LIN {X 0,Y 262.031,Z 234.936,A -85,B 0,C 180,E1 -18600.13,E2 -18600.13} C_VEL
LIN {X 0,Y 263.652,Z 236.702,A -85,B 0,C 180,E1 -18600.64,E2 -18600.64} C_VEL
LIN {X 0,Y 266.299,Z 240.265,A -85,B 0,C 180,E1 -18601.481,E2 -18601.481} C_VEL
LIN {X 0,Y 273.867,Z 250.905,A -85,B 0,C 180,E1 -18603.757,E2 -18603.757} C_VEL
LIN {X 0,Y 283.8,Z 265.428,A -85,B 0,C 180,E1 -18606.486,E2 -18606.486} C_VEL
LIN {X 0,Y 294.582,Z 283.095,A -85,B 0,C 180,E1 -18609.207,E2 -18609.207} C_VEL
LIN {X 0,Y 301.927,Z 296.558,A -85,B 0,C 180,E1 -18610.957,E2 -18610.957} C_VEL
LIN {X 0,Y 295.132,Z 420.047,A -85,B 0,C 180,E1 -18613.929,E2 -18613.929} C_VEL
LIN {X 0,Y 293.462,Z 436.562,A -85,B 0,C 180,E1 -18614.548,E2 -18614.548} C_VEL
LIN {X 0,Y 291.234,Z 452.816,A -85,B 0,C 180,E1 -18615.411,E2 -18615.411} C_VEL
LIN {X 0,Y 288.511,Z 468.704,A -85,B 0,C 180,E1 -18616.529,E2 -18616.529} C_VEL
LIN {X 0,Y 285.326,Z 484.199,A -85,B 0,C 180,E1 -18617.914,E2 -18617.914} C_VEL
LIN {X 0,Y 281.734,Z 499.193,A -85,B 0,C 180,E1 -18619.58,E2 -18619.58} C_VEL
LIN {X 0,Y 277.76,Z 513.776,A -85,B 0,C 180,E1 -18621.583,E2 -18621.583} C_VEL
LIN {X 0,Y 273.902,Z 526.637,A -85,B 0,C 180,E1 -18623.739,E2 -18623.739} C_VEL
LIN {X 0,Y 269.966,Z 539.09,A -85,B 0,C 180,E1 -18626.268,E2 -18626.268} C_VEL
LIN {X 0,Y 266.441,Z 549.708,A -85,B 0,C 180,E1 -18628.866,E2 -18628.866} C_VEL
LIN {X 0,Y 263.361,Z 558.846,A -85,B 0,C 180,E1 -18631.529,E2 -18631.529} C_VEL
LIN {X 0,Y 260.495,Z 567.585,A -85,B 0,C 180,E1 -18634.642,E2 -18634.642} C_VEL
LIN {X 0,Y 258.128,Z 574.885,A -85,B 0,C 180,E1 -18637.824,E2 -18637.824} C_VEL
LIN {X 0,Y 256.372,Z 580.903,A -85,B 0,C 180,E1 -18641.063,E2 -18641.063} C_VEL
LIN {X 0,Y 255.118,Z 585.718,A -85,B 0,C 180,E1 -18644.355,E2 -18644.355} C_VEL
LIN {X 0,Y 254.241,Z 589.354,A -85,B 0,C 180,E1 -18647.702,E2 -18647.702} C_VEL
LIN {X 0,Y 253.781,Z 591.936,A -85,B 0,C 180,E1 -18651.1,E2 -18651.1} C_VEL
LIN {X 0,Y 253.539,Z 593.385,A -85,B 0,C 180,E1 -18654.568,E2 -18654.568} C_VEL
LIN {X 0,Y 253.58,Z 593.677,A -85,B 0,C 180,E1 -18658.108,E2 -18658.108} C_VEL
LIN {X 0,Y 253.912,Z 592.8,A -85,B 0,C 180,E1 -18661.728,E2 -18661.728} C_VEL
LIN {X 0,Y 254.646,Z 590.631,A -85,B 0,C 180,E1 -18665.42,E2 -18665.42} C_VEL
LIN {X 0,Y 255.905,Z 587.007,A -85,B 0,C 180,E1 -18669.171,E2 -18669.171} C_VEL
LIN {X 0,Y 257.498,Z 582.534,A -85,B 0,C 180,E1 -18672.53,E2 -18672.53} C_VEL
LIN {X 0,Y 259.761,Z 576.753,A -85,B 0,C 180,E1 -18675.906,E2 -18675.906} C_VEL
LIN {X 0,Y 262.976,Z 568.994,A -85,B 0,C 180,E1 -18679.453,E2 -18679.453} C_VEL
LIN {X 0,Y 266.826,Z 559.99,A -85,B 0,C 180,E1 -18682.714,E2 -18682.714} C_VEL
LIN {X 0,Y 270.696,Z 550.732,A -85,B 0,C 180,E1 -18685.442,E2 -18685.442} C_VEL
LIN {X 0,Y 275.191,Z 539.733,A -85,B 0,C 180,E1 -18688.118,E2 -18688.118} C_VEL
LIN {X 0,Y 279.707,Z 527.975,A -85,B 0,C 180,E1 -18690.481,E2 -18690.481} C_VEL
LIN {X 0,Y 284.292,Z 515.315,A -85,B 0,C 180,E1 -18692.58,E2 -18692.58} C_VEL
LIN {X 0,Y 288.929,Z 500.772,A -85,B 0,C 180,E1 -18694.558,E2 -18694.558} C_VEL
LIN {X 0,Y 292.994,Z 486.399,A -85,B 0,C 180,E1 -18696.132,E2 -18696.132} C_VEL
LIN {X 0,Y 296.725,Z 471.185,A -85,B 0,C 180,E1 -18697.474,E2 -18697.474} C_VEL
LIN {X 0,Y 299.894,Z 455.605,A -85,B 0,C 180,E1 -18698.562,E2 -18698.562} C_VEL
LIN {X 0,Y 302.505,Z 439.495,A -85,B 0,C 180,E1 -18699.42,E2 -18699.42} C_VEL
LIN {X 0,Y 304.524,Z 422.953,A -85,B 0,C 180,E1 -18700.038,E2 -18700.038} C_VEL
LIN {X 0,Y 307.609,Z 376.909,A -85,B 0,C 180,E1 -18701.178,E2 -18701.178} C_VEL
LIN {X 0,Y 307.523,Z 371.142,A -85,B 0,C 180,E1 -18701.419,E2 -18701.419} C_VEL
LIN {X 0,Y 305.147,Z 352.683,A -85,B 0,C 180,E1 -18702.697,E2 -18702.697} C_VEL
LIN {X 0,Y 305.135,Z 346.914,A -85,B 0,C 180,E1 -18702.932,E2 -18702.932} C_VEL
LIN {X 0,Y 307.991,Z 305.516,A -85,B 0,C 180,E1 -18703.919,E2 -18703.919} C_VEL
LIN {X 0,Y 303.595,Z 297.18,A -85,B 0,C 180,E1 -18705.428,E2 -18705.428} C_VEL
LIN {X 0,Y 298.427,Z 288.369,A -85,B 0,C 180,E1 -18707.322,E2 -18707.322} C_VEL
LIN {X 0,Y 292.108,Z 278.333,A -85,B 0,C 180,E1 -18709.899,E2 -18709.899} C_VEL
LIN {X 0,Y 288.353,Z 273.077,A -85,B 0,C 180,E1 -18711.591,E2 -18711.591} C_VEL
LIN {X 0,Y 285.651,Z 269.277,A -85,B 0,C 180,E1 -18712.934,E2 -18712.934} C_VEL
LIN {X 0,Y 282.696,Z 265.155,A -85,B 0,C 180,E1 -18714.519,E2 -18714.519} C_VEL
LIN {X 0,Y 279.765,Z 261.171,A -85,B 0,C 180,E1 -18716.295,E2 -18716.295} C_VEL
LIN {X 0,Y 276.977,Z 258.061,A -85,B 0,C 180,E1 -18718.139,E2 -18718.139} C_VEL
LIN {X 0,Y 275.666,Z 255.828,A -85,B 0,C 180,E1 -18719.178,E2 -18719.178} C_VEL
LIN {X 0,Y 273.124,Z 252.893,A -85,B 0,C 180,E1 -18721.366,E2 -18721.366} C_VEL
LIN {X 0,Y 272.174,Z 250.924,A -85,B 0,C 180,E1 -18722.397,E2 -18722.397} C_VEL
LIN {X 0,Y 269.161,Z 249.059,A -85,B 0,C 180,E1 -18725.995,E2 -18725.995} C_VEL
LIN {X 0,Y 267.506,Z 245.335,A -85,B 0,C 180,E1 -18730.597,E2 -18730.597} C_VEL
LIN {X 0,Y 267.455,Z 245.381,A -85,B 0,C 180,E1 -18734.829,E2 -18734.829} C_VEL
LIN {X 0,Y 269.144,Z 249.233,A -85,B 0,C 180,E1 -18739.645,E2 -18739.645} C_VEL
LIN {X 0,Y 271.78,Z 251.227,A -85,B 0,C 180,E1 -18742.917,E2 -18742.917} C_VEL
LIN {X 0,Y 273.593,Z 254.335,A -85,B 0,C 180,E1 -18744.799,E2 -18744.799} C_VEL
LIN {X 0,Y 276.027,Z 256.619,A -85,B 0,C 180,E1 -18746.766,E2 -18746.766} C_VEL
LIN {X 0,Y 278.612,Z 260.377,A -85,B 0,C 180,E1 -18748.638,E2 -18748.638} C_VEL
LIN {X 0,Y 280.09,Z 262,A -85,B 0,C 180,E1 -18749.576,E2 -18749.576} C_VEL
LIN {X 0,Y 284.743,Z 268.846,A -85,B 0,C 180,E1 -18752.279,E2 -18752.279} C_VEL
LIN {X 0,Y 288.411,Z 274.538,A -85,B 0,C 180,E1 -18754.152,E2 -18754.152} C_VEL
LIN {X 0,Y 292.215,Z 280.878,A -85,B 0,C 180,E1 -18755.911,E2 -18755.911} C_VEL
LIN {X 0,Y 297.089,Z 289.527,A -85,B 0,C 180,E1 -18757.956,E2 -18757.956} C_VEL
LIN {X 0,Y 302.308,Z 299.658,A -85,B 0,C 180,E1 -18759.962,E2 -18759.962} C_VEL
LIN {X 0,Y 307.047,Z 309.971,A -85,B 0,C 180,E1 -18761.661,E2 -18761.661} C_VEL
LIN {X 0,Y 307.643,Z 311.372,A -85,B 0,C 180,E1 -18761.87,E2 -18761.87} C_VEL
LIN {X 0,Y 301.033,Z 409.803,A -85,B 0,C 180,E1 -18764.234,E2 -18764.234} C_VEL
LIN {X 0,Y 299.152,Z 435.069,A -85,B 0,C 180,E1 -18764.894,E2 -18764.894} C_VEL
LIN {X 0,Y 296.911,Z 451.91,A -85,B 0,C 180,E1 -18765.521,E2 -18765.521} C_VEL
LIN {X 0,Y 293.976,Z 467.817,A -85,B 0,C 180,E1 -18766.347,E2 -18766.347} C_VEL
LIN {X 0,Y 290.572,Z 482.839,A -85,B 0,C 180,E1 -18767.374,E2 -18767.374} C_VEL
LIN {X 0,Y 286.439,Z 498.519,A -85,B 0,C 180,E1 -18768.747,E2 -18768.747} C_VEL
LIN {X 0,Y 281.831,Z 513.372,A -85,B 0,C 180,E1 -18770.353,E2 -18770.353} C_VEL
LIN {X 0,Y 277.266,Z 526.892,A -85,B 0,C 180,E1 -18772.176,E2 -18772.176} C_VEL
LIN {X 0,Y 272.027,Z 540.712,A -85,B 0,C 180,E1 -18774.459,E2 -18774.459} C_VEL
LIN {X 0,Y 267.105,Z 552.94,A -85,B 0,C 180,E1 -18776.955,E2 -18776.955} C_VEL
LIN {X 0,Y 262.933,Z 563.126,A -85,B 0,C 180,E1 -18779.48,E2 -18779.48} C_VEL
LIN {X 0,Y 259.086,Z 572.103,A -85,B 0,C 180,E1 -18782.101,E2 -18782.101} C_VEL
LIN {X 0,Y 254.99,Z 581.757,A -85,B 0,C 180,E1 -18785.581,E2 -18785.581} C_VEL
LIN {X 0,Y 251.535,Z 590.443,A -85,B 0,C 180,E1 -18789.559,E2 -18789.559} C_VEL
LIN {X 0,Y 249.09,Z 597.237,A -85,B 0,C 180,E1 -18793.612,E2 -18793.612} C_VEL
LIN {X 0,Y 247.847,Z 601.386,A -85,B 0,C 180,E1 -18796.889,E2 -18796.889} C_VEL
LIN {X 0,Y 247.104,Z 604.584,A -85,B 0,C 180,E1 -18800.175,E2 -18800.175} C_VEL
LIN {X 0,Y 246.856,Z 606.689,A -85,B 0,C 180,E1 -18803.462,E2 -18803.462} C_VEL
LIN {X 0,Y 246.839,Z 607.899,A -85,B 0,C 180,E1 -18806.736,E2 -18806.736} C_VEL
LIN {X 0,Y 246.983,Z 608.047,A -85,B 0,C 180,E1 -18810,E2 -18810} C_VEL
LIN {X 0,Y 246.868,Z 607.28,A -85,B 0,C 180,E1 -18813.264,E2 -18813.264} C_VEL
LIN {X 0,Y 246.859,Z 605.423,A -85,B 0,C 180,E1 -18816.539,E2 -18816.539} C_VEL
LIN {X 0,Y 247.096,Z 602.604,A -85,B 0,C 180,E1 -18819.826,E2 -18819.826} C_VEL
LIN {X 0,Y 248.074,Z 597.527,A -85,B 0,C 180,E1 -18823.934,E2 -18823.934} C_VEL
LIN {X 0,Y 249.357,Z 592.125,A -85,B 0,C 180,E1 -18827.214,E2 -18827.214} C_VEL
LIN {X 0,Y 251.252,Z 585.487,A -85,B 0,C 180,E1 -18830.466,E2 -18830.466} C_VEL
LIN {X 0,Y 253.657,Z 577.952,A -85,B 0,C 180,E1 -18833.512,E2 -18833.512} C_VEL
LIN {X 0,Y 257.031,Z 567.882,A -85,B 0,C 180,E1 -18836.818,E2 -18836.818} C_VEL
LIN {X 0,Y 260.52,Z 557.897,A -85,B 0,C 180,E1 -18839.494,E2 -18839.494} C_VEL
LIN {X 0,Y 263.756,Z 547.897,A -85,B 0,C 180,E1 -18841.783,E2 -18841.783} C_VEL
LIN {X 0,Y 267.797,Z 535.618,A -85,B 0,C 180,E1 -18844.122,E2 -18844.122} C_VEL
LIN {X 0,Y 271.945,Z 522.038,A -85,B 0,C 180,E1 -18846.24,E2 -18846.24} C_VEL
LIN {X 0,Y 275.628,Z 508.654,A -85,B 0,C 180,E1 -18847.962,E2 -18847.962} C_VEL
LIN {X 0,Y 279.266,Z 494.431,A -85,B 0,C 180,E1 -18849.453,E2 -18849.453} C_VEL
LIN {X 0,Y 282.538,Z 479.102,A -85,B 0,C 180,E1 -18850.765,E2 -18850.765} C_VEL
LIN {X 0,Y 285.543,Z 462.08,A -85,B 0,C 180,E1 -18851.884,E2 -18851.884} C_VEL
LIN {X 0,Y 287.982,Z 444.871,A -85,B 0,C 180,E1 -18852.686,E2 -18852.686} C_VEL
LIN {X 0,Y 289.505,Z 429.304,A -85,B 0,C 180,E1 -18853.181,E2 -18853.181} C_VEL
LIN {X 0,Y 296.362,Z 306.373,A -85,B 0,C 180,E1 -18856.178,E2 -18856.178} C_VEL
LIN {X 0,Y 288.532,Z 290.028,A -85,B 0,C 180,E1 -18858.18,E2 -18858.18} C_VEL
LIN {X 0,Y 280.5,Z 274.97,A -85,B 0,C 180,E1 -18860.348,E2 -18860.348} C_VEL
LIN {X 0,Y 272.954,Z 261.95,A -85,B 0,C 180,E1 -18862.512,E2 -18862.512} C_VEL
LIN {X 0,Y 266.916,Z 252.198,A -85,B 0,C 180,E1 -18864.362,E2 -18864.362} C_VEL
LIN {X 0,Y 262.167,Z 245.051,A -85,B 0,C 180,E1 -18865.891,E2 -18865.891} C_VEL
LIN {X 0,Y 259.448,Z 241.346,A -85,B 0,C 180,E1 -18866.791,E2 -18866.791} C_VEL
LIN {X 0,Y 256.707,Z 237.544,A -85,B 0,C 180,E1 -18867.735,E2 -18867.735} C_VEL
LIN {X 0,Y 253.618,Z 233.906,A -85,B 0,C 180,E1 -18868.812,E2 -18868.812} C_VEL
LIN {X 0,Y 252.501,Z 232.01,A -85,B 0,C 180,E1 -18869.24,E2 -18869.24} C_VEL
LIN {X 0,Y 250.243,Z 229.914,A -85,B 0,C 180,E1 -18870.039,E2 -18870.039} C_VEL
LIN {X 0,Y 249.171,Z 227.301,A -85,B 0,C 180,E1 -18870.514,E2 -18870.514} C_VEL
LIN {X 0,Y 249.076,Z 226.767,A -85,B 0,C 180,E1 -18870.596,E2 -18870.596} C_VEL
LIN {X 0,Y 249.15,Z 226.733,A -85,B 0,C 180,E1 -18874.969,E2 -18874.969} C_VEL
LIN {X 0,Y 249.093,Z 226.751,A -85,B 0,C 180,E1 -18878.602,E2 -18878.602} C_VEL
LIN {X 0,Y 249.195,Z 226.752,A -85,B 0,C 180,E1 -18883.619,E2 -18883.619} C_VEL
LIN {X 0,Y 249.224,Z 226.704,A -85,B 0,C 180,E1 -18888.615,E2 -18888.615} C_VEL
LIN {X 0,Y 249.441,Z 226.724,A -85,B 0,C 180,E1 -18891.902,E2 -18891.902} C_VEL
LIN {X 0,Y 249.287,Z 226.704,A -85,B 0,C 180,E1 -18895.148,E2 -18895.148} C_VEL
LIN {X 0,Y 249.673,Z 226.648,A -85,B 0,C 180,E1 -18898.387,E2 -18898.387} C_VEL
LIN {X 0,Y 249.674,Z 226.697,A -85,B 0,C 180,E1 -18901.613,E2 -18901.613} C_VEL
LIN {X 0,Y 249.439,Z 226.705,A -85,B 0,C 180,E1 -18906.718,E2 -18906.718} C_VEL
LIN {X 0,Y 249.343,Z 226.728,A -85,B 0,C 180,E1 -18909.736,E2 -18909.736} C_VEL
LIN {X 0,Y 249.205,Z 226.752,A -85,B 0,C 180,E1 -18914.703,E2 -18914.703} C_VEL
LIN {X 0,Y 249.139,Z 226.734,A -85,B 0,C 180,E1 -18918.077,E2 -18918.077} C_VEL
LIN {X 0,Y 249.087,Z 226.767,A -85,B 0,C 180,E1 -18921.518,E2 -18921.518} C_VEL
LIN {X 0,Y 249.131,Z 226.735,A -85,B 0,C 180,E1 -18925.482,E2 -18925.482} C_VEL
LIN {X 0,Y 249.087,Z 226.771,A -85,B 0,C 180,E1 -18928.995,E2 -18928.995} C_VEL
LIN {X 0,Y 249.03,Z 226.751,A -85,B 0,C 180,E1 -18932.426,E2 -18932.426} C_VEL
LIN {X 0,Y 249.047,Z 226.766,A -85,B 0,C 180,E1 -18936.342,E2 -18936.342} C_VEL
LIN {X 0,Y 249.006,Z 226.779,A -85,B 0,C 180,E1 -18940.478,E2 -18940.478} C_VEL
LIN {X 0,Y 248.992,Z 226.766,A -85,B 0,C 180,E1 -18944.881,E2 -18944.881} C_VEL
LIN {X 0,Y 249.015,Z 226.773,A -85,B 0,C 180,E1 -18947.363,E2 -18947.363} C_VEL
LIN {X 0,Y 249.043,Z 226.769,A -85,B 0,C 180,E1 -18952.2,E2 -18952.2} C_VEL
LIN {X 0,Y 249.04,Z 226.774,A -85,B 0,C 180,E1 -18955.931,E2 -18955.931} C_VEL
LIN {X 0,Y 249.82,Z 229.243,A -85,B 0,C 180,E1 -18956.312,E2 -18956.312} C_VEL
LIN {X 0,Y 251.534,Z 231.358,A -85,B 0,C 180,E1 -18956.952,E2 -18956.952} C_VEL
LIN {X 0,Y 252.919,Z 232.5,A -85,B 0,C 180,E1 -18957.431,E2 -18957.431} C_VEL
LIN {X 0,Y 254.879,Z 235.654,A -85,B 0,C 180,E1 -18958.17,E2 -18958.17} C_VEL
LIN {X 0,Y 256.812,Z 237.703,A -85,B 0,C 180,E1 -18958.826,E2 -18958.826} C_VEL
LIN {X 0,Y 259.44,Z 241.277,A -85,B 0,C 180,E1 -18959.724,E2 -18959.724} C_VEL
LIN {X 0,Y 264.351,Z 247.934,A -85,B 0,C 180,E1 -18961.322,E2 -18961.322} C_VEL
LIN {X 0,Y 271.132,Z 257.534,A -85,B 0,C 180,E1 -18963.396,E2 -18963.396} C_VEL
LIN {X 0,Y 280.204,Z 271.03,A -85,B 0,C 180,E1 -18965.95,E2 -18965.95} C_VEL
LIN {X 0,Y 290.389,Z 287.903,A -85,B 0,C 180,E1 -18968.604,E2 -18968.604} C_VEL
LIN {X 0,Y 296.481,Z 299.015,A -85,B 0,C 180,E1 -18970.096,E2 -18970.096} C_VEL
LIN {X 0,Y 289.59,Z 420.591,A -85,B 0,C 180,E1 -18973.068,E2 -18973.068} C_VEL
LIN {X 0,Y 287.767,Z 437.863,A -85,B 0,C 180,E1 -18973.734,E2 -18973.734} C_VEL
LIN {X 0,Y 285.368,Z 454.472,A -85,B 0,C 180,E1 -18974.649,E2 -18974.649} C_VEL
LIN {X 0,Y 282.549,Z 470.029,A -85,B 0,C 180,E1 -18975.781,E2 -18975.781} C_VEL
LIN {X 0,Y 279.48,Z 484.488,A -85,B 0,C 180,E1 -18977.104,E2 -18977.104} C_VEL
LIN {X 0,Y 275.759,Z 499.477,A -85,B 0,C 180,E1 -18978.794,E2 -18978.794} C_VEL
LIN {X 0,Y 271.899,Z 513.198,A -85,B 0,C 180,E1 -18980.703,E2 -18980.703} C_VEL
LIN {X 0,Y 267.953,Z 525.923,A -85,B 0,C 180,E1 -18982.843,E2 -18982.843} C_VEL
LIN {X 0,Y 263.832,Z 538.529,A -85,B 0,C 180,E1 -18985.416,E2 -18985.416} C_VEL
LIN {X 0,Y 260.187,Z 549.178,A -85,B 0,C 180,E1 -18988.039,E2 -18988.039} C_VEL
LIN {X 0,Y 256.875,Z 558.489,A -85,B 0,C 180,E1 -18990.783,E2 -18990.783} C_VEL
LIN {X 0,Y 254.101,Z 566.572,A -85,B 0,C 180,E1 -18993.676,E2 -18993.676} C_VEL
LIN {X 0,Y 251.966,Z 573.039,A -85,B 0,C 180,E1 -18996.405,E2 -18996.405} C_VEL
LIN {X 0,Y 249.78,Z 579.919,A -85,B 0,C 180,E1 -19000.008,E2 -19000.008} C_VEL
LIN {X 0,Y 248.437,Z 584.554,A -85,B 0,C 180,E1 -19003.079,E2 -19003.079} C_VEL
LIN {X 0,Y 247.423,Z 588.606,A -85,B 0,C 180,E1 -19006.501,E2 -19006.501} C_VEL
LIN {X 0,Y 246.813,Z 591.473,A -85,B 0,C 180,E1 -19010.003,E2 -19010.003} C_VEL
LIN {X 0,Y 246.5,Z 593.256,A -85,B 0,C 180,E1 -19013.525,E2 -19013.525} C_VEL
LIN {X 0,Y 246.47,Z 593.959,A -85,B 0,C 180,E1 -19017.143,E2 -19017.143} C_VEL
LIN {X 0,Y 246.772,Z 593.275,A -85,B 0,C 180,E1 -19021.308,E2 -19021.308} C_VEL
LIN {X 0,Y 247.347,Z 591.61,A -85,B 0,C 180,E1 -19024.629,E2 -19024.629} C_VEL
LIN {X 0,Y 248.521,Z 588.471,A -85,B 0,C 180,E1 -19028.472,E2 -19028.472} C_VEL
LIN {X 0,Y 250.303,Z 583.834,A -85,B 0,C 180,E1 -19032.365,E2 -19032.365} C_VEL
LIN {X 0,Y 252.908,Z 577.541,A -85,B 0,C 180,E1 -19036.26,E2 -19036.26} C_VEL
LIN {X 0,Y 255.621,Z 571.302,A -85,B 0,C 180,E1 -19039.275,E2 -19039.275} C_VEL
LIN {X 0,Y 259.171,Z 563.406,A -85,B 0,C 180,E1 -19042.407,E2 -19042.407} C_VEL
LIN {X 0,Y 263.047,Z 554.718,A -85,B 0,C 180,E1 -19045.24,E2 -19045.24} C_VEL
LIN {X 0,Y 267.499,Z 544.525,A -85,B 0,C 180,E1 -19047.951,E2 -19047.951} C_VEL
LIN {X 0,Y 272.168,Z 533.037,A -85,B 0,C 180,E1 -19050.494,E2 -19050.494} C_VEL
LIN {X 0,Y 277.286,Z 519.862,A -85,B 0,C 180,E1 -19052.857,E2 -19052.857} C_VEL
LIN {X 0,Y 281.815,Z 506.845,A -85,B 0,C 180,E1 -19054.785,E2 -19054.785} C_VEL
LIN {X 0,Y 286.126,Z 493.17,A -85,B 0,C 180,E1 -19056.437,E2 -19056.437} C_VEL
LIN {X 0,Y 290.151,Z 478.375,A -85,B 0,C 180,E1 -19057.891,E2 -19057.891} C_VEL
LIN {X 0,Y 293.792,Z 462.5,A -85,B 0,C 180,E1 -19059.135,E2 -19059.135} C_VEL
LIN {X 0,Y 296.806,Z 446.047,A -85,B 0,C 180,E1 -19060.131,E2 -19060.131} C_VEL
LIN {X 0,Y 299.107,Z 430.324,A -85,B 0,C 180,E1 -19060.814,E2 -19060.814} C_VEL
LIN {X 0,Y 300.702,Z 413.397,A -85,B 0,C 180,E1 -19061.331,E2 -19061.331} C_VEL
LIN {X 0,Y 305.135,Z 346.914,A -85,B 0,C 180,E1 -19062.932,E2 -19062.932} C_VEL
LIN {X 0,Y 305.117,Z 341.14,A -85,B 0,C 180,E1 -19063.172,E2 -19063.172} C_VEL
LIN {X 0,Y 302.957,Z 322.696,A -85,B 0,C 180,E1 -19064.495,E2 -19064.495} C_VEL
LIN {X 0,Y 303.017,Z 316.921,A -85,B 0,C 180,E1 -19064.727,E2 -19064.727} C_VEL
LIN {X 0,Y 303.577,Z 308.469,A -85,B 0,C 180,E1 -19064.943,E2 -19064.943} C_VEL
LIN {X 0,Y 297.727,Z 297.627,A -85,B 0,C 180,E1 -19067.094,E2 -19067.094} C_VEL
LIN {X 0,Y 291.284,Z 287.028,A -85,B 0,C 180,E1 -19069.722,E2 -19069.722} C_VEL
LIN {X 0,Y 287.001,Z 280.473,A -85,B 0,C 180,E1 -19071.689,E2 -19071.689} C_VEL
LIN {X 0,Y 283.314,Z 275.274,A -85,B 0,C 180,E1 -19073.567,E2 -19073.567} C_VEL
LIN {X 0,Y 280.767,Z 271.594,A -85,B 0,C 180,E1 -19075.004,E2 -19075.004} C_VEL
LIN {X 0,Y 277.936,Z 267.662,A -85,B 0,C 180,E1 -19076.788,E2 -19076.788} C_VEL
LIN {X 0,Y 275.207,Z 264.392,A -85,B 0,C 180,E1 -19078.691,E2 -19078.691} C_VEL
LIN {X 0,Y 274.093,Z 262.494,A -85,B 0,C 180,E1 -19079.611,E2 -19079.611} C_VEL
LIN {X 0,Y 271.623,Z 259.443,A -85,B 0,C 180,E1 -19081.853,E2 -19081.853} C_VEL
LIN {X 0,Y 270.795,Z 257.779,A -85,B 0,C 180,E1 -19082.788,E2 -19082.788} C_VEL
LIN {X 0,Y 268.104,Z 256.047,A -85,B 0,C 180,E1 -19086.14,E2 -19086.14} C_VEL
LIN {X 0,Y 266.541,Z 252.403,A -85,B 0,C 180,E1 -19090.636,E2 -19090.636} C_VEL
LIN {X 0,Y 266.469,Z 252.375,A -85,B 0,C 180,E1 -19094.639,E2 -19094.639} C_VEL
LIN {X 0,Y 268.102,Z 256.239,A -85,B 0,C 180,E1 -19099.525,E2 -19099.525} C_VEL
LIN {X 0,Y 270.449,Z 258.043,A -85,B 0,C 180,E1 -19102.554,E2 -19102.554} C_VEL
LIN {X 0,Y 272.334,Z 261.239,A -85,B 0,C 180,E1 -19104.565,E2 -19104.565} C_VEL
LIN {X 0,Y 274.434,Z 263.232,A -85,B 0,C 180,E1 -19106.324,E2 -19106.324} C_VEL
LIN {X 0,Y 277.07,Z 267.119,A -85,B 0,C 180,E1 -19108.308,E2 -19108.308} C_VEL
LIN {X 0,Y 278.306,Z 268.529,A -85,B 0,C 180,E1 -19109.118,E2 -19109.118} C_VEL
LIN {X 0,Y 282.522,Z 274.891,A -85,B 0,C 180,E1 -19111.685,E2 -19111.685} C_VEL
LIN {X 0,Y 286.095,Z 280.674,A -85,B 0,C 180,E1 -19113.589,E2 -19113.589} C_VEL
LIN {X 0,Y 289.17,Z 285.918,A -85,B 0,C 180,E1 -19115.088,E2 -19115.088} C_VEL
LIN {X 0,Y 293.972,Z 294.702,A -85,B 0,C 180,E1 -19117.221,E2 -19117.221} C_VEL
LIN {X 0,Y 299.004,Z 304.731,A -85,B 0,C 180,E1 -19119.256,E2 -19119.256} C_VEL
LIN {X 0,Y 303.342,Z 314.363,A -85,B 0,C 180,E1 -19120.882,E2 -19120.882} C_VEL
LIN {X 0,Y 294.908,Z 432.361,A -85,B 0,C 180,E1 -19123.756,E2 -19123.756} C_VEL
LIN {X 0,Y 292.717,Z 449.242,A -85,B 0,C 180,E1 -19124.365,E2 -19124.365} C_VEL
LIN {X 0,Y 289.958,Z 464.391,A -85,B 0,C 180,E1 -19125.107,E2 -19125.107} C_VEL
LIN {X 0,Y 286.429,Z 480.071,A -85,B 0,C 180,E1 -19126.121,E2 -19126.121} C_VEL
LIN {X 0,Y 282.62,Z 494.63,A -85,B 0,C 180,E1 -19127.342,E2 -19127.342} C_VEL
LIN {X 0,Y 277.936,Z 509.588,A -85,B 0,C 180,E1 -19128.896,E2 -19128.896} C_VEL
LIN {X 0,Y 273.365,Z 522.759,A -85,B 0,C 180,E1 -19130.595,E2 -19130.595} C_VEL
LIN {X 0,Y 268.623,Z 535.26,A -85,B 0,C 180,E1 -19132.535,E2 -19132.535} C_VEL
LIN {X 0,Y 264.064,Z 546.425,A -85,B 0,C 180,E1 -19134.63,E2 -19134.63} C_VEL
LIN {X 0,Y 259.165,Z 557.798,A -85,B 0,C 180,E1 -19137.209,E2 -19137.209} C_VEL
LIN {X 0,Y 254.369,Z 568.531,A -85,B 0,C 180,E1 -19140.178,E2 -19140.178} C_VEL
LIN {X 0,Y 250.246,Z 577.75,A -85,B 0,C 180,E1 -19143.299,E2 -19143.299} C_VEL
LIN {X 0,Y 246.88,Z 585.475,A -85,B 0,C 180,E1 -19146.514,E2 -19146.514} C_VEL
LIN {X 0,Y 244.195,Z 591.877,A -85,B 0,C 180,E1 -19149.797,E2 -19149.797} C_VEL
LIN {X 0,Y 242.119,Z 597.41,A -85,B 0,C 180,E1 -19153.313,E2 -19153.313} C_VEL
LIN {X 0,Y 240.864,Z 601.283,A -85,B 0,C 180,E1 -19156.502,E2 -19156.502} C_VEL
LIN {X 0,Y 240.04,Z 604.442,A -85,B 0,C 180,E1 -19159.883,E2 -19159.883} C_VEL
LIN {X 0,Y 239.767,Z 606.529,A -85,B 0,C 180,E1 -19163.267,E2 -19163.267} C_VEL
LIN {X 0,Y 239.744,Z 607.702,A -85,B 0,C 180,E1 -19166.639,E2 -19166.639} C_VEL
LIN {X 0,Y 239.913,Z 607.831,A -85,B 0,C 180,E1 -19170,E2 -19170} C_VEL
LIN {X 0,Y 239.774,Z 607.025,A -85,B 0,C 180,E1 -19173.361,E2 -19173.361} C_VEL
LIN {X 0,Y 239.821,Z 606.225,A -85,B 0,C 180,E1 -19175.044,E2 -19175.044} C_VEL
LIN {X 0,Y 239.872,Z 603.837,A -85,B 0,C 180,E1 -19178.424,E2 -19178.424} C_VEL
LIN {X 0,Y 240.328,Z 600.46,A -85,B 0,C 180,E1 -19181.812,E2 -19181.812} C_VEL
LIN {X 0,Y 241.675,Z 594.851,A -85,B 0,C 180,E1 -19185.88,E2 -19185.88} C_VEL
LIN {X 0,Y 243.38,Z 588.545,A -85,B 0,C 180,E1 -19189.395,E2 -19189.395} C_VEL
LIN {X 0,Y 245.775,Z 581.2,A -85,B 0,C 180,E1 -19192.708,E2 -19192.708} C_VEL
LIN {X 0,Y 248.772,Z 572.38,A -85,B 0,C 180,E1 -19195.969,E2 -19195.969} C_VEL
LIN {X 0,Y 252.593,Z 561.814,A -85,B 0,C 180,E1 -19199.138,E2 -19199.138} C_VEL
LIN {X 0,Y 256.238,Z 551.194,A -85,B 0,C 180,E1 -19201.761,E2 -19201.761} C_VEL
LIN {X 0,Y 260.141,Z 539.855,A -85,B 0,C 180,E1 -19204.096,E2 -19204.096} C_VEL
LIN {X 0,Y 264.271,Z 527.153,A -85,B 0,C 180,E1 -19206.279,E2 -19206.279} C_VEL
LIN {X 0,Y 268.62,Z 512.782,A -85,B 0,C 180,E1 -19208.289,E2 -19208.289} C_VEL
LIN {X 0,Y 272.422,Z 498.392,A -85,B 0,C 180,E1 -19209.921,E2 -19209.921} C_VEL
LIN {X 0,Y 276.057,Z 482.886,A -85,B 0,C 180,E1 -19211.325,E2 -19211.325} C_VEL
LIN {X 0,Y 279.119,Z 466.976,A -85,B 0,C 180,E1 -19212.463,E2 -19212.463} C_VEL
LIN {X 0,Y 281.564,Z 451.74,A -85,B 0,C 180,E1 -19213.286,E2 -19213.286} C_VEL
LIN {X 0,Y 283.655,Z 434.645,A -85,B 0,C 180,E1 -19213.927,E2 -19213.927} C_VEL
LIN {X 0,Y 287.302,Z 371.522,A -85,B 0,C 180,E1 -19215.53,E2 -19215.53} C_VEL
LIN {X 0,Y 290.939,Z 308.736,A -85,B 0,C 180,E1 -19217.067,E2 -19217.067} C_VEL
LIN {X 0,Y 283.914,Z 293.977,A -85,B 0,C 180,E1 -19218.934,E2 -19218.934} C_VEL
LIN {X 0,Y 276.164,Z 279.314,A -85,B 0,C 180,E1 -19221.1,E2 -19221.1} C_VEL
LIN {X 0,Y 269.039,Z 266.863,A -85,B 0,C 180,E1 -19223.226,E2 -19223.226} C_VEL
LIN {X 0,Y 263.188,Z 257.265,A -85,B 0,C 180,E1 -19225.079,E2 -19225.079} C_VEL
LIN {X 0,Y 258.352,Z 249.977,A -85,B 0,C 180,E1 -19226.69,E2 -19226.69} C_VEL
LIN {X 0,Y 255.752,Z 246.482,A -85,B 0,C 180,E1 -19227.579,E2 -19227.579} C_VEL
LIN {X 0,Y 252.776,Z 242.472,A -85,B 0,C 180,E1 -19228.638,E2 -19228.638} C_VEL
LIN {X 0,Y 250.118,Z 238.942,A -85,B 0,C 180,E1 -19229.617,E2 -19229.617} C_VEL
LIN {X 0,Y 248.959,Z 237.619,A -85,B 0,C 180,E1 -19230.046,E2 -19230.046} C_VEL
LIN {X 0,Y 246.642,Z 234.687,A -85,B 0,C 180,E1 -19230.944,E2 -19230.944} C_VEL
LIN {X 0,Y 245.802,Z 233.041,A -85,B 0,C 180,E1 -19231.309,E2 -19231.309} C_VEL
LIN {X 0,Y 243.556,Z 231.25,A -85,B 0,C 180,E1 -19232.154,E2 -19232.154} C_VEL
LIN {X 0,Y 242.234,Z 228.656,A -85,B 0,C 180,E1 -19232.751,E2 -19232.751} C_VEL
LIN {X 0,Y 242.037,Z 227.621,A -85,B 0,C 180,E1 -19232.903,E2 -19232.903} C_VEL
LIN {X 0,Y 242.056,Z 227.63,A -85,B 0,C 180,E1 -19236.016,E2 -19236.016} C_VEL
LIN {X 0,Y 242.025,Z 227.614,A -85,B 0,C 180,E1 -19239.607,E2 -19239.607} C_VEL
LIN {X 0,Y 242.115,Z 227.628,A -85,B 0,C 180,E1 -19243.316,E2 -19243.316} C_VEL
LIN {X 0,Y 242.134,Z 227.6,A -85,B 0,C 180,E1 -19246.573,E2 -19246.573} C_VEL
LIN {X 0,Y 242.388,Z 227.599,A -85,B 0,C 180,E1 -19251.664,E2 -19251.664} C_VEL
LIN {X 0,Y 242.415,Z 227.597,A -85,B 0,C 180,E1 -19253.341,E2 -19253.341} C_VEL
LIN {X 0,Y 242.633,Z 227.523,A -85,B 0,C 180,E1 -19258.34,E2 -19258.34} C_VEL
LIN {X 0,Y 242.635,Z 227.574,A -85,B 0,C 180,E1 -19261.66,E2 -19261.66} C_VEL
LIN {X 0,Y 242.42,Z 227.58,A -85,B 0,C 180,E1 -19266.69,E2 -19266.69} C_VEL
LIN {X 0,Y 242.267,Z 227.604,A -85,B 0,C 180,E1 -19270.024,E2 -19270.024} C_VEL
LIN {X 0,Y 242.166,Z 227.63,A -85,B 0,C 180,E1 -19275.141,E2 -19275.141} C_VEL
LIN {X 0,Y 242.072,Z 227.611,A -85,B 0,C 180,E1 -19278.624,E2 -19278.624} C_VEL
LIN {X 0,Y 242.013,Z 227.651,A -85,B 0,C 180,E1 -19282.18,E2 -19282.18} C_VEL
LIN {X 0,Y 242.066,Z 227.615,A -85,B 0,C 180,E1 -19285.838,E2 -19285.838} C_VEL
LIN {X 0,Y 242.031,Z 227.645,A -85,B 0,C 180,E1 -19289.58,E2 -19289.58} C_VEL
LIN {X 0,Y 241.98,Z 227.638,A -85,B 0,C 180,E1 -19293.493,E2 -19293.493} C_VEL
LIN {X 0,Y 241.988,Z 227.631,A -85,B 0,C 180,E1 -19297.582,E2 -19297.582} C_VEL
LIN {X 0,Y 241.933,Z 227.656,A -85,B 0,C 180,E1 -19301.923,E2 -19301.923} C_VEL
LIN {X 0,Y 241.932,Z 227.663,A -85,B 0,C 180,E1 -19306.572,E2 -19306.572} C_VEL
LIN {X 0,Y 241.995,Z 227.654,A -85,B 0,C 180,E1 -19311.64,E2 -19311.64} C_VEL
LIN {X 0,Y 242.007,Z 227.631,A -85,B 0,C 180,E1 -19313.613,E2 -19313.613} C_VEL
LIN {X 0,Y 242.841,Z 230.251,A -85,B 0,C 180,E1 -19314.065,E2 -19314.065} C_VEL
LIN {X 0,Y 244.62,Z 232.316,A -85,B 0,C 180,E1 -19314.788,E2 -19314.788} C_VEL
LIN {X 0,Y 246.005,Z 233.437,A -85,B 0,C 180,E1 -19315.309,E2 -19315.309} C_VEL
LIN {X 0,Y 247.819,Z 236.494,A -85,B 0,C 180,E1 -19316.056,E2 -19316.056} C_VEL
LIN {X 0,Y 250.001,Z 238.742,A -85,B 0,C 180,E1 -19316.854,E2 -19316.854} C_VEL
LIN {X 0,Y 252.623,Z 242.292,A -85,B 0,C 180,E1 -19317.827,E2 -19317.827} C_VEL
LIN {X 0,Y 253.937,Z 243.955,A -85,B 0,C 180,E1 -19318.298,E2 -19318.298} C_VEL
LIN {X 0,Y 258.355,Z 249.931,A -85,B 0,C 180,E1 -19319.828,E2 -19319.828} C_VEL
LIN {X 0,Y 263.589,Z 257.098,A -85,B 0,C 180,E1 -19321.533,E2 -19321.533} C_VEL
LIN {X 0,Y 273.699,Z 272.015,A -85,B 0,C 180,E1 -19324.577,E2 -19324.577} C_VEL
LIN {X 0,Y 283.097,Z 287.351,A -85,B 0,C 180,E1 -19327.163,E2 -19327.163} C_VEL
LIN {X 0,Y 291.075,Z 301.655,A -85,B 0,C 180,E1 -19329.218,E2 -19329.218} C_VEL
LIN {X 0,Y 284.114,Z 420.909,A -85,B 0,C 180,E1 -19332.175,E2 -19332.175} C_VEL
LIN {X 0,Y 282.224,Z 438.164,A -85,B 0,C 180,E1 -19332.846,E2 -19332.846} C_VEL
LIN {X 0,Y 279.77,Z 454.714,A -85,B 0,C 180,E1 -19333.771,E2 -19333.771} C_VEL
LIN {X 0,Y 276.905,Z 470.097,A -85,B 0,C 180,E1 -19334.903,E2 -19334.903} C_VEL
LIN {X 0,Y 273.682,Z 484.76,A -85,B 0,C 180,E1 -19336.259,E2 -19336.259} C_VEL
LIN {X 0,Y 269.831,Z 499.758,A -85,B 0,C 180,E1 -19337.973,E2 -19337.973} C_VEL
LIN {X 0,Y 265.843,Z 513.477,A -85,B 0,C 180,E1 -19339.913,E2 -19339.913} C_VEL
LIN {X 0,Y 261.444,Z 527.177,A -85,B 0,C 180,E1 -19342.275,E2 -19342.275} C_VEL
LIN {X 0,Y 257.211,Z 539.611,A -85,B 0,C 180,E1 -19344.905,E2 -19344.905} C_VEL
LIN {X 0,Y 253.197,Z 550.784,A -85,B 0,C 180,E1 -19347.778,E2 -19347.778} C_VEL
LIN {X 0,Y 249.644,Z 560.484,A -85,B 0,C 180,E1 -19350.806,E2 -19350.806} C_VEL
LIN {X 0,Y 246.6,Z 569.05,A -85,B 0,C 180,E1 -19354.066,E2 -19354.066} C_VEL
LIN {X 0,Y 244.088,Z 576.205,A -85,B 0,C 180,E1 -19357.444,E2 -19357.444} C_VEL
LIN {X 0,Y 242.206,Z 582.028,A -85,B 0,C 180,E1 -19360.871,E2 -19360.871} C_VEL
LIN {X 0,Y 240.923,Z 586.701,A -85,B 0,C 180,E1 -19364.356,E2 -19364.356} C_VEL
LIN {X 0,Y 240.211,Z 589.413,A -85,B 0,C 180,E1 -19367.012,E2 -19367.012} C_VEL
LIN {X 0,Y 239.631,Z 592.137,A -85,B 0,C 180,E1 -19370.605,E2 -19370.605} C_VEL
LIN {X 0,Y 239.366,Z 593.735,A -85,B 0,C 180,E1 -19374.469,E2 -19374.469} C_VEL
LIN {X 0,Y 239.428,Z 594.104,A -85,B 0,C 180,E1 -19378.286,E2 -19378.286} C_VEL
LIN {X 0,Y 239.731,Z 593.405,A -85,B 0,C 180,E1 -19381.849,E2 -19381.849} C_VEL
LIN {X 0,Y 240.518,Z 591.324,A -85,B 0,C 180,E1 -19385.76,E2 -19385.76} C_VEL
LIN {X 0,Y 241.926,Z 587.874,A -85,B 0,C 180,E1 -19389.724,E2 -19389.724} C_VEL
LIN {X 0,Y 243.989,Z 582.912,A -85,B 0,C 180,E1 -19393.733,E2 -19393.733} C_VEL
LIN {X 0,Y 246.126,Z 578.114,A -85,B 0,C 180,E1 -19396.74,E2 -19396.74} C_VEL
LIN {X 0,Y 249.321,Z 571.189,A -85,B 0,C 180,E1 -19400.185,E2 -19400.185} C_VEL
LIN {X 0,Y 253.348,Z 562.72,A -85,B 0,C 180,E1 -19403.558,E2 -19403.558} C_VEL
LIN {X 0,Y 257.436,Z 554.1,A -85,B 0,C 180,E1 -19406.37,E2 -19406.37} C_VEL
LIN {X 0,Y 262.106,Z 543.899,A -85,B 0,C 180,E1 -19409.094,E2 -19409.094} C_VEL
LIN {X 0,Y 267.174,Z 531.879,A -85,B 0,C 180,E1 -19411.739,E2 -19411.739} C_VEL
LIN {X 0,Y 272.192,Z 519.37,A -85,B 0,C 180,E1 -19413.964,E2 -19413.964} C_VEL
LIN {X 0,Y 277.043,Z 505.882,A -85,B 0,C 180,E1 -19415.955,E2 -19415.955} C_VEL
LIN {X 0,Y 281.342,Z 492.657,A -85,B 0,C 180,E1 -19417.556,E2 -19417.556} C_VEL
LIN {X 0,Y 285.843,Z 476.597,A -85,B 0,C 180,E1 -19419.113,E2 -19419.113} C_VEL
LIN {X 0,Y 289.557,Z 460.568,A -85,B 0,C 180,E1 -19420.327,E2 -19420.327} C_VEL
LIN {X 0,Y 292.52,Z 444.255,A -85,B 0,C 180,E1 -19421.284,E2 -19421.284} C_VEL
LIN {X 0,Y 294.812,Z 428.232,A -85,B 0,C 180,E1 -19421.946,E2 -19421.946} C_VEL
LIN {X 0,Y 296.499,Z 409.306,A -85,B 0,C 180,E1 -19422.49,E2 -19422.49} C_VEL
LIN {X 0,Y 303.017,Z 316.921,A -85,B 0,C 180,E1 -19424.727,E2 -19424.727} C_VEL
LIN {X 0,Y 302.739,Z 314.026,A -85,B 0,C 180,E1 -19424.928,E2 -19424.928} C_VEL
LIN {X 0,Y 301.508,Z 311.266,A -85,B 0,C 180,E1 -19425.385,E2 -19425.385} C_VEL
LIN {X 0,Y 300.117,Z 309.526,A -85,B 0,C 180,E1 -19425.851,E2 -19425.851} C_VEL
LIN {X 0,Y 295.927,Z 305.22,A -85,B 0,C 180,E1 -19427.28,E2 -19427.28} C_VEL
LIN {X 0,Y 295.151,Z 303.898,A -85,B 0,C 180,E1 -19427.583,E2 -19427.583} C_VEL
LIN {X 0,Y 289.274,Z 293.739,A -85,B 0,C 180,E1 -19430.077,E2 -19430.077} C_VEL
LIN {X 0,Y 284.435,Z 286.216,A -85,B 0,C 180,E1 -19432.389,E2 -19432.389} C_VEL
LIN {X 0,Y 280.621,Z 280.692,A -85,B 0,C 180,E1 -19434.431,E2 -19434.431} C_VEL
LIN {X 0,Y 278.597,Z 277.682,A -85,B 0,C 180,E1 -19435.66,E2 -19435.66} C_VEL
LIN {X 0,Y 276.283,Z 274.312,A -85,B 0,C 180,E1 -19437.185,E2 -19437.185} C_VEL
LIN {X 0,Y 273.556,Z 270.909,A -85,B 0,C 180,E1 -19439.175,E2 -19439.175} C_VEL
LIN {X 0,Y 272.61,Z 269.227,A -85,B 0,C 180,E1 -19440,E2 -19440} C_VEL
LIN {X 0,Y 270.263,Z 266.197,A -85,B 0,C 180,E1 -19442.221,E2 -19442.221} C_VEL
LIN {X 0,Y 269.433,Z 264.654,A -85,B 0,C 180,E1 -19443.177,E2 -19443.177} C_VEL
LIN {X 0,Y 266.967,Z 262.936,A -85,B 0,C 180,E1 -19446.424,E2 -19446.424} C_VEL
LIN {X 0,Y 265.575,Z 259.473,A -85,B 0,C 180,E1 -19450.675,E2 -19450.675} C_VEL
LIN {X 0,Y 265.487,Z 259.369,A -85,B 0,C 180,E1 -19454.447,E2 -19454.447} C_VEL
LIN {X 0,Y 266.986,Z 263.152,A -85,B 0,C 180,E1 -19459.275,E2 -19459.275} C_VEL
LIN {X 0,Y 269.171,Z 264.928,A -85,B 0,C 180,E1 -19462.236,E2 -19462.236} C_VEL
LIN {X 0,Y 271.121,Z 268.19,A -85,B 0,C 180,E1 -19464.368,E2 -19464.368} C_VEL
LIN {X 0,Y 273.019,Z 270.173,A -85,B 0,C 180,E1 -19466.022,E2 -19466.022} C_VEL
LIN {X 0,Y 275.661,Z 273.97,A -85,B 0,C 180,E1 -19468.056,E2 -19468.056} C_VEL
LIN {X 0,Y 276.876,Z 275.645,A -85,B 0,C 180,E1 -19468.89,E2 -19468.89} C_VEL
LIN {X 0,Y 280.39,Z 281.092,A -85,B 0,C 180,E1 -19471.12,E2 -19471.12} C_VEL
LIN {X 0,Y 284.176,Z 287.372,A -85,B 0,C 180,E1 -19473.207,E2 -19473.207} C_VEL
LIN {X 0,Y 288.048,Z 294.305,A -85,B 0,C 180,E1 -19475.14,E2 -19475.14} C_VEL
LIN {X 0,Y 292.493,Z 303.023,A -85,B 0,C 180,E1 -19477.16,E2 -19477.16} C_VEL
LIN {X 0,Y 297.186,Z 312.858,A -85,B 0,C 180,E1 -19479.098,E2 -19479.098} C_VEL
LIN {X 0,Y 299.06,Z 317.23,A -85,B 0,C 180,E1 -19479.84,E2 -19479.84} C_VEL
LIN {X 0,Y 290.515,Z 432.436,A -85,B 0,C 180,E1 -19482.664,E2 -19482.664} C_VEL
LIN {X 0,Y 288.172,Z 449.71,A -85,B 0,C 180,E1 -19483.296,E2 -19483.296} C_VEL
LIN {X 0,Y 285.332,Z 464.599,A -85,B 0,C 180,E1 -19484.036,E2 -19484.036} C_VEL
LIN {X 0,Y 281.935,Z 479.246,A -85,B 0,C 180,E1 -19484.984,E2 -19484.984} C_VEL
LIN {X 0,Y 278.445,Z 492.144,A -85,B 0,C 180,E1 -19486.046,E2 -19486.046} C_VEL
LIN {X 0,Y 274.092,Z 506.119,A -85,B 0,C 180,E1 -19487.448,E2 -19487.448} C_VEL
LIN {X 0,Y 269.477,Z 519.322,A -85,B 0,C 180,E1 -19489.062,E2 -19489.062} C_VEL
LIN {X 0,Y 263.848,Z 533.729,A -85,B 0,C 180,E1 -19491.249,E2 -19491.249} C_VEL
LIN {X 0,Y 258.281,Z 546.764,A -85,B 0,C 180,E1 -19493.714,E2 -19493.714} C_VEL
LIN {X 0,Y 252.941,Z 558.563,A -85,B 0,C 180,E1 -19496.465,E2 -19496.465} C_VEL
LIN {X 0,Y 248.174,Z 568.694,A -85,B 0,C 180,E1 -19499.355,E2 -19499.355} C_VEL
LIN {X 0,Y 243.852,Z 577.839,A -85,B 0,C 180,E1 -19502.541,E2 -19502.541} C_VEL
LIN {X 0,Y 240.3,Z 585.513,A -85,B 0,C 180,E1 -19505.83,E2 -19505.83} C_VEL
LIN {X 0,Y 237.456,Z 591.86,A -85,B 0,C 180,E1 -19509.197,E2 -19509.197} C_VEL
LIN {X 0,Y 235.122,Z 597.633,A -85,B 0,C 180,E1 -19513.039,E2 -19513.039} C_VEL
LIN {X 0,Y 233.899,Z 601.195,A -85,B 0,C 180,E1 -19516.092,E2 -19516.092} C_VEL
LIN {X 0,Y 232.994,Z 604.305,A -85,B 0,C 180,E1 -19519.574,E2 -19519.574} C_VEL
LIN {X 0,Y 232.668,Z 606.369,A -85,B 0,C 180,E1 -19523.061,E2 -19523.061} C_VEL
LIN {X 0,Y 232.652,Z 607.505,A -85,B 0,C 180,E1 -19526.537,E2 -19526.537} C_VEL
LIN {X 0,Y 232.822,Z 607.616,A -85,B 0,C 180,E1 -19530.001,E2 -19530.001} C_VEL
LIN {X 0,Y 232.684,Z 606.769,A -85,B 0,C 180,E1 -19533.464,E2 -19533.464} C_VEL
LIN {X 0,Y 232.73,Z 605.969,A -85,B 0,C 180,E1 -19535.198,E2 -19535.198} C_VEL
LIN {X 0,Y 232.808,Z 603.539,A -85,B 0,C 180,E1 -19538.682,E2 -19538.682} C_VEL
LIN {X 0,Y 233.312,Z 600.133,A -85,B 0,C 180,E1 -19542.173,E2 -19542.173} C_VEL
LIN {X 0,Y 234.466,Z 595.523,A -85,B 0,C 180,E1 -19545.651,E2 -19545.651} C_VEL
LIN {X 0,Y 236.079,Z 589.778,A -85,B 0,C 180,E1 -19549.115,E2 -19549.115} C_VEL
LIN {X 0,Y 238.431,Z 582.748,A -85,B 0,C 180,E1 -19552.532,E2 -19552.532} C_VEL
LIN {X 0,Y 241.413,Z 574.199,A -85,B 0,C 180,E1 -19555.892,E2 -19555.892} C_VEL
LIN {X 0,Y 245.188,Z 564.003,A -85,B 0,C 180,E1 -19559.162,E2 -19559.162} C_VEL
LIN {X 0,Y 248.54,Z 555.131,A -85,B 0,C 180,E1 -19561.542,E2 -19561.542} C_VEL
LIN {X 0,Y 252.842,Z 542.985,A -85,B 0,C 180,E1 -19564.254,E2 -19564.254} C_VEL
LIN {X 0,Y 256.981,Z 530.744,A -85,B 0,C 180,E1 -19566.5,E2 -19566.5} C_VEL
LIN {X 0,Y 261.352,Z 517.069,A -85,B 0,C 180,E1 -19568.562,E2 -19568.562} C_VEL
LIN {X 0,Y 265.232,Z 503.624,A -85,B 0,C 180,E1 -19570.231,E2 -19570.231} C_VEL
LIN {X 0,Y 269.122,Z 488.406,A -85,B 0,C 180,E1 -19571.753,E2 -19571.753} C_VEL
LIN {X 0,Y 272.472,Z 472.682,A -85,B 0,C 180,E1 -19572.993,E2 -19572.993} C_VEL
LIN {X 0,Y 275.233,Z 456.835,A -85,B 0,C 180,E1 -19573.952,E2 -19573.952} C_VEL
LIN {X 0,Y 277.619,Z 439.61,A -85,B 0,C 180,E1 -19574.688,E2 -19574.688} C_VEL
LIN {X 0,Y 278.954,Z 422.941,A -85,B 0,C 180,E1 -19575.197,E2 -19575.197} C_VEL
LIN {X 0,Y 285.632,Z 311.246,A -85,B 0,C 180,E1 -19577.966,E2 -19577.966} C_VEL
LIN {X 0,Y 278.675,Z 296.509,A -85,B 0,C 180,E1 -19579.904,E2 -19579.904} C_VEL
LIN {X 0,Y 270.582,Z 281.218,A -85,B 0,C 180,E1 -19582.268,E2 -19582.268} C_VEL
LIN {X 0,Y 261.681,Z 265.856,A -85,B 0,C 180,E1 -19585.083,E2 -19585.083} C_VEL
LIN {X 0,Y 255.348,Z 255.943,A -85,B 0,C 180,E1 -19587.243,E2 -19587.243} C_VEL
LIN {X 0,Y 252.259,Z 251.776,A -85,B 0,C 180,E1 -19588.332,E2 -19588.332} C_VEL
LIN {X 0,Y 249.47,Z 248.041,A -85,B 0,C 180,E1 -19589.354,E2 -19589.354} C_VEL
LIN {X 0,Y 246.285,Z 243.79,A -85,B 0,C 180,E1 -19590.578,E2 -19590.578} C_VEL
LIN {X 0,Y 243.615,Z 240.418,A -85,B 0,C 180,E1 -19591.635,E2 -19591.635} C_VEL
LIN {X 0,Y 242.524,Z 238.926,A -85,B 0,C 180,E1 -19592.084,E2 -19592.084} C_VEL
LIN {X 0,Y 239.99,Z 236.099,A -85,B 0,C 180,E1 -19593.123,E2 -19593.123} C_VEL
LIN {X 0,Y 238.786,Z 233.903,A -85,B 0,C 180,E1 -19593.684,E2 -19593.684} C_VEL
LIN {X 0,Y 236.277,Z 231.766,A -85,B 0,C 180,E1 -19594.753,E2 -19594.753} C_VEL
LIN {X 0,Y 235.176,Z 229.404,A -85,B 0,C 180,E1 -19595.327,E2 -19595.327} C_VEL
LIN {X 0,Y 235.012,Z 228.498,A -85,B 0,C 180,E1 -19595.485,E2 -19595.485} C_VEL
LIN {X 0,Y 235.005,Z 228.496,A -85,B 0,C 180,E1 -19598.969,E2 -19598.969} C_VEL
LIN {X 0,Y 235.08,Z 228.517,A -85,B 0,C 180,E1 -19604.391,E2 -19604.391} C_VEL
LIN {X 0,Y 235.185,Z 228.458,A -85,B 0,C 180,E1 -19609.671,E2 -19609.671} C_VEL
LIN {X 0,Y 235.365,Z 228.478,A -85,B 0,C 180,E1 -19613.14,E2 -19613.14} C_VEL
LIN {X 0,Y 235.593,Z 228.398,A -85,B 0,C 180,E1 -19618.291,E2 -19618.291} C_VEL
LIN {X 0,Y 235.594,Z 228.452,A -85,B 0,C 180,E1 -19621.709,E2 -19621.709} C_VEL
LIN {X 0,Y 235.373,Z 228.46,A -85,B 0,C 180,E1 -19626.86,E2 -19626.86} C_VEL
LIN {X 0,Y 235.214,Z 228.477,A -85,B 0,C 180,E1 -19630.328,E2 -19630.328} C_VEL
LIN {X 0,Y 235.113,Z 228.51,A -85,B 0,C 180,E1 -19635.606,E2 -19635.606} C_VEL
LIN {X 0,Y 235.008,Z 228.491,A -85,B 0,C 180,E1 -19639.206,E2 -19639.206} C_VEL
LIN {X 0,Y 234.961,Z 228.526,A -85,B 0,C 180,E1 -19642.883,E2 -19642.883} C_VEL
LIN {X 0,Y 234.971,Z 228.504,A -85,B 0,C 180,E1 -19646.657,E2 -19646.657} C_VEL
LIN {X 0,Y 234.932,Z 228.515,A -85,B 0,C 180,E1 -19650.568,E2 -19650.568} C_VEL
LIN {X 0,Y 234.93,Z 228.532,A -85,B 0,C 180,E1 -19654.638,E2 -19654.638} C_VEL
LIN {X 0,Y 234.942,Z 228.509,A -85,B 0,C 180,E1 -19658.944,E2 -19658.944} C_VEL
LIN {X 0,Y 234.879,Z 228.518,A -85,B 0,C 180,E1 -19663.488,E2 -19663.488} C_VEL
LIN {X 0,Y 234.885,Z 228.541,A -85,B 0,C 180,E1 -19666.513,E2 -19666.513} C_VEL
LIN {X 0,Y 234.942,Z 228.653,A -85,B 0,C 180,E1 -19671.056,E2 -19671.056} C_VEL
LIN {X 0,Y 235.721,Z 230.997,A -85,B 0,C 180,E1 -19671.502,E2 -19671.502} C_VEL
LIN {X 0,Y 237.744,Z 233.332,A -85,B 0,C 180,E1 -19672.403,E2 -19672.403} C_VEL
LIN {X 0,Y 239.087,Z 234.305,A -85,B 0,C 180,E1 -19672.954,E2 -19672.954} C_VEL
LIN {X 0,Y 240.968,Z 237.465,A -85,B 0,C 180,E1 -19673.811,E2 -19673.811} C_VEL
LIN {X 0,Y 243.234,Z 239.778,A -85,B 0,C 180,E1 -19674.726,E2 -19674.726} C_VEL
LIN {X 0,Y 245.573,Z 243.114,A -85,B 0,C 180,E1 -19675.682,E2 -19675.682} C_VEL
LIN {X 0,Y 247.231,Z 245.014,A -85,B 0,C 180,E1 -19676.311,E2 -19676.311} C_VEL
LIN {X 0,Y 251.378,Z 250.552,A -85,B 0,C 180,E1 -19677.867,E2 -19677.867} C_VEL
LIN {X 0,Y 255.446,Z 256.025,A -85,B 0,C 180,E1 -19679.309,E2 -19679.309} C_VEL
LIN {X 0,Y 261.083,Z 264.001,A -85,B 0,C 180,E1 -19681.196,E2 -19681.196} C_VEL
LIN {X 0,Y 270.154,Z 277.587,A -85,B 0,C 180,E1 -19683.995,E2 -19683.995} C_VEL
LIN {X 0,Y 278.456,Z 291.229,A -85,B 0,C 180,E1 -19686.361,E2 -19686.361} C_VEL
LIN {X 0,Y 285.745,Z 304.332,A -85,B 0,C 180,E1 -19688.313,E2 -19688.313} C_VEL
LIN {X 0,Y 278.69,Z 421.091,A -85,B 0,C 180,E1 -19691.244,E2 -19691.244} C_VEL
LIN {X 0,Y 276.757,Z 438.323,A -85,B 0,C 180,E1 -19691.923,E2 -19691.923} C_VEL
LIN {X 0,Y 274.41,Z 453.634,A -85,B 0,C 180,E1 -19692.774,E2 -19692.774} C_VEL
LIN {X 0,Y 271.604,Z 468.714,A -85,B 0,C 180,E1 -19693.872,E2 -19693.872} C_VEL
LIN {X 0,Y 268.371,Z 483.315,A -85,B 0,C 180,E1 -19695.207,E2 -19695.207} C_VEL
LIN {X 0,Y 264.318,Z 498.56,A -85,B 0,C 180,E1 -19696.938,E2 -19696.938} C_VEL
LIN {X 0,Y 260.216,Z 512.484,A -85,B 0,C 180,E1 -19698.905,E2 -19698.905} C_VEL
LIN {X 0,Y 255.807,Z 525.819,A -85,B 0,C 180,E1 -19701.19,E2 -19701.19} C_VEL
LIN {X 0,Y 251.818,Z 537.348,A -85,B 0,C 180,E1 -19703.59,E2 -19703.59} C_VEL
LIN {X 0,Y 247.709,Z 548.381,A -85,B 0,C 180,E1 -19706.339,E2 -19706.339} C_VEL
LIN {X 0,Y 243.651,Z 558.983,A -85,B 0,C 180,E1 -19709.586,E2 -19709.586} C_VEL
LIN {X 0,Y 240.34,Z 567.817,A -85,B 0,C 180,E1 -19712.933,E2 -19712.933} C_VEL
LIN {X 0,Y 237.973,Z 574.351,A -85,B 0,C 180,E1 -19715.932,E2 -19715.932} C_VEL
LIN {X 0,Y 235.878,Z 580.35,A -85,B 0,C 180,E1 -19719.278,E2 -19719.278} C_VEL
LIN {X 0,Y 234.27,Z 585.568,A -85,B 0,C 180,E1 -19723.002,E2 -19723.002} C_VEL
LIN {X 0,Y 233.418,Z 588.59,A -85,B 0,C 180,E1 -19725.722,E2 -19725.722} C_VEL
LIN {X 0,Y 232.676,Z 591.591,A -85,B 0,C 180,E1 -19729.405,E2 -19729.405} C_VEL
LIN {X 0,Y 232.303,Z 593.546,A -85,B 0,C 180,E1 -19733.159,E2 -19733.159} C_VEL
LIN {X 0,Y 232.24,Z 594.33,A -85,B 0,C 180,E1 -19736.995,E2 -19736.995} C_VEL
LIN {X 0,Y 232.505,Z 593.933,A -85,B 0,C 180,E1 -19740.92,E2 -19740.92} C_VEL
LIN {X 0,Y 233.233,Z 592.312,A -85,B 0,C 180,E1 -19744.925,E2 -19744.925} C_VEL
LIN {X 0,Y 234.514,Z 589.344,A -85,B 0,C 180,E1 -19749,E2 -19749} C_VEL
LIN {X 0,Y 236.487,Z 584.838,A -85,B 0,C 180,E1 -19753.118,E2 -19753.118} C_VEL
LIN {X 0,Y 239.36,Z 578.718,A -85,B 0,C 180,E1 -19757.225,E2 -19757.225} C_VEL
LIN {X 0,Y 242.267,Z 572.809,A -85,B 0,C 180,E1 -19760.342,E2 -19760.342} C_VEL
LIN {X 0,Y 246.274,Z 564.912,A -85,B 0,C 180,E1 -19763.722,E2 -19763.722} C_VEL
LIN {X 0,Y 251.157,Z 555.072,A -85,B 0,C 180,E1 -19767.083,E2 -19767.083} C_VEL
LIN {X 0,Y 256.632,Z 543.591,A -85,B 0,C 180,E1 -19770.212,E2 -19770.212} C_VEL
LIN {X 0,Y 261.987,Z 531.538,A -85,B 0,C 180,E1 -19772.868,E2 -19772.868} C_VEL
LIN {X 0,Y 267.22,Z 518.953,A -85,B 0,C 180,E1 -19775.115,E2 -19775.115} C_VEL
LIN {X 0,Y 272.169,Z 505.629,A -85,B 0,C 180,E1 -19777.079,E2 -19777.079} C_VEL
LIN {X 0,Y 276.976,Z 491.052,A -85,B 0,C 180,E1 -19778.824,E2 -19778.824} C_VEL
LIN {X 0,Y 281.23,Z 476.418,A -85,B 0,C 180,E1 -19780.223,E2 -19780.223} C_VEL
LIN {X 0,Y 285.11,Z 460.257,A -85,B 0,C 180,E1 -19781.445,E2 -19781.445} C_VEL
LIN {X 0,Y 287.97,Z 444.945,A -85,B 0,C 180,E1 -19782.35,E2 -19782.35} C_VEL
LIN {X 0,Y 290.494,Z 427.932,A -85,B 0,C 180,E1 -19783.055,E2 -19783.055} C_VEL
LIN {X 0,Y 292.264,Z 408.373,A -85,B 0,C 180,E1 -19783.613,E2 -19783.613} C_VEL
LIN {X 0,Y 299.295,Z 311.679,A -85,B 0,C 180,E1 -19785.976,E2 -19785.976} C_VEL
LIN {X 0,Y 295.151,Z 303.898,A -85,B 0,C 180,E1 -19787.583,E2 -19787.583} C_VEL
LIN {X 0,Y 292.969,Z 300.688,A -85,B 0,C 180,E1 -19788.442,E2 -19788.442} C_VEL
LIN {X 0,Y 290.449,Z 298.528,A -85,B 0,C 180,E1 -19789.406,E2 -19789.406} C_VEL
LIN {X 0,Y 283.74,Z 294.176,A -85,B 0,C 180,E1 -19792.189,E2 -19792.189} C_VEL
LIN {X 0,Y 282.346,Z 292.557,A -85,B 0,C 180,E1 -19792.878,E2 -19792.878} C_VEL
LIN {X 0,Y 277.269,Z 284.767,A -85,B 0,C 180,E1 -19795.821,E2 -19795.821} C_VEL
LIN {X 0,Y 274.485,Z 280.828,A -85,B 0,C 180,E1 -19797.692,E2 -19797.692} C_VEL
LIN {X 0,Y 271.783,Z 277.143,A -85,B 0,C 180,E1 -19799.792,E2 -19799.792} C_VEL
LIN {X 0,Y 270.894,Z 275.673,A -85,B 0,C 180,E1 -19800.617,E2 -19800.617} C_VEL
LIN {X 0,Y 268.731,Z 272.582,A -85,B 0,C 180,E1 -19802.81,E2 -19802.81} C_VEL
LIN {X 0,Y 268.268,Z 271.6,A -85,B 0,C 180,E1 -19803.379,E2 -19803.379} C_VEL
LIN {X 0,Y 265.864,Z 269.86,A -85,B 0,C 180,E1 -19806.663,E2 -19806.663} C_VEL
LIN {X 0,Y 264.612,Z 266.524,A -85,B 0,C 180,E1 -19810.715,E2 -19810.715} C_VEL
LIN {X 0,Y 264.51,Z 266.362,A -85,B 0,C 180,E1 -19814.254,E2 -19814.254} C_VEL
LIN {X 0,Y 266.007,Z 270.209,A -85,B 0,C 180,E1 -19819.253,E2 -19819.253} C_VEL
LIN {X 0,Y 267.963,Z 271.953,A -85,B 0,C 180,E1 -19821.986,E2 -19821.986} C_VEL
LIN {X 0,Y 270.038,Z 275.278,A -85,B 0,C 180,E1 -19824.289,E2 -19824.289} C_VEL
LIN {X 0,Y 271.565,Z 277,A -85,B 0,C 180,E1 -19825.666,E2 -19825.666} C_VEL
LIN {X 0,Y 274.371,Z 280.947,A -85,B 0,C 180,E1 -19827.88,E2 -19827.88} C_VEL
LIN {X 0,Y 278.222,Z 287.076,A -85,B 0,C 180,E1 -19830.474,E2 -19830.474} C_VEL
LIN {X 0,Y 282.133,Z 293.82,A -85,B 0,C 180,E1 -19832.743,E2 -19832.743} C_VEL
LIN {X 0,Y 286.229,Z 301.593,A -85,B 0,C 180,E1 -19834.871,E2 -19834.871} C_VEL
LIN {X 0,Y 291.22,Z 311.871,A -85,B 0,C 180,E1 -19837.191,E2 -19837.191} C_VEL
LIN {X 0,Y 294.922,Z 320.224,A -85,B 0,C 180,E1 -19838.766,E2 -19838.766} C_VEL
LIN {X 0,Y 286.241,Z 432.626,A -85,B 0,C 180,E1 -19841.543,E2 -19841.543} C_VEL
LIN {X 0,Y 283.711,Z 450.464,A -85,B 0,C 180,E1 -19842.199,E2 -19842.199} C_VEL
LIN {X 0,Y 280.79,Z 465.081,A -85,B 0,C 180,E1 -19842.938,E2 -19842.938} C_VEL
LIN {X 0,Y 277.025,Z 480.535,A -85,B 0,C 180,E1 -19843.958,E2 -19843.958} C_VEL
LIN {X 0,Y 272.938,Z 494.924,A -85,B 0,C 180,E1 -19845.181,E2 -19845.181} C_VEL
LIN {X 0,Y 267.988,Z 509.712,A -85,B 0,C 180,E1 -19846.756,E2 -19846.756} C_VEL
LIN {X 0,Y 263.014,Z 522.85,A -85,B 0,C 180,E1 -19848.48,E2 -19848.48} C_VEL
LIN {X 0,Y 257.487,Z 536.143,A -85,B 0,C 180,E1 -19850.611,E2 -19850.611} C_VEL
LIN {X 0,Y 251.826,Z 548.818,A -85,B 0,C 180,E1 -19853.129,E2 -19853.129} C_VEL
LIN {X 0,Y 246.801,Z 559.306,A -85,B 0,C 180,E1 -19855.671,E2 -19855.671} C_VEL
LIN {X 0,Y 242.045,Z 568.859,A -85,B 0,C 180,E1 -19858.491,E2 -19858.491} C_VEL
LIN {X 0,Y 237.518,Z 577.937,A -85,B 0,C 180,E1 -19861.744,E2 -19861.744} C_VEL
LIN {X 0,Y 233.748,Z 585.583,A -85,B 0,C 180,E1 -19865.107,E2 -19865.107} C_VEL
LIN {X 0,Y 230.099,Z 593.3,A -85,B 0,C 180,E1 -19869.437,E2 -19869.437} C_VEL
LIN {X 0,Y 227.644,Z 599.228,A -85,B 0,C 180,E1 -19873.869,E2 -19873.869} C_VEL
LIN {X 0,Y 226.324,Z 602.753,A -85,B 0,C 180,E1 -19877.446,E2 -19877.446} C_VEL
LIN {X 0,Y 225.723,Z 605.347,A -85,B 0,C 180,E1 -19881.045,E2 -19881.045} C_VEL
LIN {X 0,Y 225.553,Z 607.157,A -85,B 0,C 180,E1 -19885.622,E2 -19885.622} C_VEL
LIN {X 0,Y 225.654,Z 607.505,A -85,B 0,C 180,E1 -19888.216,E2 -19888.216} C_VEL
LIN {X 0,Y 225.734,Z 607.4,A -85,B 0,C 180,E1 -19890.001,E2 -19890.001} C_VEL
LIN {X 0,Y 225.597,Z 606.513,A -85,B 0,C 180,E1 -19893.573,E2 -19893.573} C_VEL
LIN {X 0,Y 225.635,Z 605.712,A -85,B 0,C 180,E1 -19895.362,E2 -19895.362} C_VEL
LIN {X 0,Y 225.728,Z 603.239,A -85,B 0,C 180,E1 -19898.956,E2 -19898.956} C_VEL
LIN {X 0,Y 226.317,Z 599.793,A -85,B 0,C 180,E1 -19902.555,E2 -19902.555} C_VEL
LIN {X 0,Y 227.541,Z 595.148,A -85,B 0,C 180,E1 -19906.14,E2 -19906.14} C_VEL
LIN {X 0,Y 229.266,Z 589.345,A -85,B 0,C 180,E1 -19909.706,E2 -19909.706} C_VEL
LIN {X 0,Y 231.77,Z 582.276,A -85,B 0,C 180,E1 -19913.216,E2 -19913.216} C_VEL
LIN {X 0,Y 235.365,Z 572.511,A -85,B 0,C 180,E1 -19917.089,E2 -19917.089} C_VEL
LIN {X 0,Y 239.501,Z 562.005,A -85,B 0,C 180,E1 -19920.41,E2 -19920.41} C_VEL
LIN {X 0,Y 243.539,Z 551.093,A -85,B 0,C 180,E1 -19923.25,E2 -19923.25} C_VEL
LIN {X 0,Y 247.575,Z 540.266,A -85,B 0,C 180,E1 -19925.587,E2 -19925.587} C_VEL
LIN {X 0,Y 252.009,Z 527.702,A -85,B 0,C 180,E1 -19927.845,E2 -19927.845} C_VEL
LIN {X 0,Y 256.65,Z 513.323,A -85,B 0,C 180,E1 -19929.938,E2 -19929.938} C_VEL
LIN {X 0,Y 260.637,Z 499.244,A -85,B 0,C 180,E1 -19931.606,E2 -19931.606} C_VEL
LIN {X 0,Y 264.479,Z 484.05,A -85,B 0,C 180,E1 -19933.047,E2 -19933.047} C_VEL
LIN {X 0,Y 267.724,Z 468.617,A -85,B 0,C 180,E1 -19934.21,E2 -19934.21} C_VEL
LIN {X 0,Y 270.51,Z 452.586,A -85,B 0,C 180,E1 -19935.117,E2 -19935.117} C_VEL
LIN {X 0,Y 272.705,Z 435.703,A -85,B 0,C 180,E1 -19935.779,E2 -19935.779} C_VEL
LIN {X 0,Y 274.551,Z 407.366,A -85,B 0,C 180,E1 -19936.561,E2 -19936.561} C_VEL
LIN {X 0,Y 280.39,Z 313.691,A -85,B 0,C 180,E1 -19938.903,E2 -19938.903} C_VEL
LIN {X 0,Y 273.175,Z 298.574,A -85,B 0,C 180,E1 -19940.986,E2 -19940.986} C_VEL
LIN {X 0,Y 265.37,Z 283.833,A -85,B 0,C 180,E1 -19943.385,E2 -19943.385} C_VEL
LIN {X 0,Y 257.82,Z 270.669,A -85,B 0,C 180,E1 -19945.879,E2 -19945.879} C_VEL
LIN {X 0,Y 251.956,Z 261.322,A -85,B 0,C 180,E1 -19947.954,E2 -19947.954} C_VEL
LIN {X 0,Y 246.319,Z 253.701,A -85,B 0,C 180,E1 -19950.047,E2 -19950.047} C_VEL
LIN {X 0,Y 243.066,Z 249.397,A -85,B 0,C 180,E1 -19951.332,E2 -19951.332} C_VEL
LIN {X 0,Y 240.255,Z 245.504,A -85,B 0,C 180,E1 -19952.5,E2 -19952.5} C_VEL
LIN {X 0,Y 237.187,Z 241.993,A -85,B 0,C 180,E1 -19953.801,E2 -19953.801} C_VEL
LIN {X 0,Y 235.927,Z 240.008,A -85,B 0,C 180,E1 -19954.392,E2 -19954.392} C_VEL
LIN {X 0,Y 233.494,Z 237.55,A -85,B 0,C 180,E1 -19955.493,E2 -19955.493} C_VEL
LIN {X 0,Y 232.095,Z 234.98,A -85,B 0,C 180,E1 -19956.227,E2 -19956.227} C_VEL
LIN {X 0,Y 229.744,Z 233.343,A -85,B 0,C 180,E1 -19957.311,E2 -19957.311} C_VEL
LIN {X 0,Y 228.351,Z 230.973,A -85,B 0,C 180,E1 -19958.066,E2 -19958.066} C_VEL
LIN {X 0,Y 227.945,Z 229.384,A -85,B 0,C 180,E1 -19958.404,E2 -19958.404} C_VEL
LIN {X 0,Y 228.023,Z 229.392,A -85,B 0,C 180,E1 -19963.895,E2 -19963.895} C_VEL
LIN {X 0,Y 228.053,Z 229.341,A -85,B 0,C 180,E1 -19967.542,E2 -19967.542} C_VEL
LIN {X 0,Y 228.249,Z 229.347,A -85,B 0,C 180,E1 -19971.144,E2 -19971.144} C_VEL
LIN {X 0,Y 228.315,Z 229.357,A -85,B 0,C 180,E1 -19972.927,E2 -19972.927} C_VEL
LIN {X 0,Y 228.551,Z 229.273,A -85,B 0,C 180,E1 -19978.238,E2 -19978.238} C_VEL
LIN {X 0,Y 228.553,Z 229.329,A -85,B 0,C 180,E1 -19981.762,E2 -19981.762} C_VEL
LIN {X 0,Y 228.323,Z 229.34,A -85,B 0,C 180,E1 -19987.072,E2 -19987.072} C_VEL
LIN {X 0,Y 228.145,Z 229.352,A -85,B 0,C 180,E1 -19990.651,E2 -19990.651} C_VEL
LIN {X 0,Y 228.064,Z 229.378,A -85,B 0,C 180,E1 -19994.272,E2 -19994.272} C_VEL
LIN {X 0,Y 228.003,Z 229.365,A -85,B 0,C 180,E1 -19997.953,E2 -19997.953} C_VEL
LIN {X 0,Y 227.93,Z 229.405,A -85,B 0,C 180,E1 -20002.329,E2 -20002.329} C_VEL
LIN {X 0,Y 227.944,Z 229.378,A -85,B 0,C 180,E1 -20006.603,E2 -20006.603} C_VEL
LIN {X 0,Y 227.909,Z 229.393,A -85,B 0,C 180,E1 -20010.296,E2 -20010.296} C_VEL
LIN {X 0,Y 227.877,Z 229.396,A -85,B 0,C 180,E1 -20013.72,E2 -20013.72} C_VEL
LIN {X 0,Y 227.843,Z 229.39,A -85,B 0,C 180,E1 -20018.091,E2 -20018.091} C_VEL
LIN {X 0,Y 227.806,Z 229.403,A -85,B 0,C 180,E1 -20022.743,E2 -20022.743} C_VEL
LIN {X 0,Y 227.808,Z 229.414,A -85,B 0,C 180,E1 -20027.257,E2 -20027.257} C_VEL
LIN {X 0,Y 227.852,Z 229.506,A -85,B 0,C 180,E1 -20028.126,E2 -20028.126} C_VEL
LIN {X 0,Y 228.66,Z 231.932,A -85,B 0,C 180,E1 -20028.646,E2 -20028.646} C_VEL
LIN {X 0,Y 230.601,Z 234.188,A -85,B 0,C 180,E1 -20029.634,E2 -20029.634} C_VEL
LIN {X 0,Y 232.203,Z 235.3,A -85,B 0,C 180,E1 -20030.372,E2 -20030.372} C_VEL
LIN {X 0,Y 234.245,Z 238.629,A -85,B 0,C 180,E1 -20031.394,E2 -20031.394} C_VEL
LIN {X 0,Y 236.466,Z 240.749,A -85,B 0,C 180,E1 -20032.365,E2 -20032.365} C_VEL
LIN {X 0,Y 238.939,Z 244.236,A -85,B 0,C 180,E1 -20033.474,E2 -20033.474} C_VEL
LIN {X 0,Y 240.508,Z 245.992,A -85,B 0,C 180,E1 -20034.129,E2 -20034.129} C_VEL
LIN {X 0,Y 243.432,Z 249.807,A -85,B 0,C 180,E1 -20035.336,E2 -20035.336} C_VEL
LIN {X 0,Y 248.839,Z 257.072,A -85,B 0,C 180,E1 -20037.428,E2 -20037.428} C_VEL
LIN {X 0,Y 254.05,Z 264.187,A -85,B 0,C 180,E1 -20039.303,E2 -20039.303} C_VEL
LIN {X 0,Y 262.514,Z 276.72,A -85,B 0,C 180,E1 -20042.124,E2 -20042.124} C_VEL
LIN {X 0,Y 270.58,Z 289.552,A -85,B 0,C 180,E1 -20044.584,E2 -20044.584} C_VEL
LIN {X 0,Y 279.369,Z 304.936,A -85,B 0,C 180,E1 -20047.07,E2 -20047.07} C_VEL
LIN {X 0,Y 280.559,Z 307.65,A -85,B 0,C 180,E1 -20047.412,E2 -20047.412} C_VEL
LIN {X 0,Y 273.334,Z 421.293,A -85,B 0,C 180,E1 -20050.277,E2 -20050.277} C_VEL
LIN {X 0,Y 271.345,Z 438.515,A -85,B 0,C 180,E1 -20050.962,E2 -20050.962} C_VEL
LIN {X 0,Y 268.736,Z 455.077,A -85,B 0,C 180,E1 -20051.907,E2 -20051.907} C_VEL
LIN {X 0,Y 265.637,Z 470.668,A -85,B 0,C 180,E1 -20053.08,E2 -20053.08} C_VEL
LIN {X 0,Y 262.277,Z 485.122,A -85,B 0,C 180,E1 -20054.457,E2 -20054.457} C_VEL
LIN {X 0,Y 258.127,Z 500.156,A -85,B 0,C 180,E1 -20056.217,E2 -20056.217} C_VEL
LIN {X 0,Y 253.885,Z 513.876,A -85,B 0,C 180,E1 -20058.22,E2 -20058.22} C_VEL
LIN {X 0,Y 249.35,Z 527.083,A -85,B 0,C 180,E1 -20060.567,E2 -20060.567} C_VEL
LIN {X 0,Y 245.251,Z 538.38,A -85,B 0,C 180,E1 -20063.004,E2 -20063.004} C_VEL
LIN {X 0,Y 241.018,Z 549.283,A -85,B 0,C 180,E1 -20065.819,E2 -20065.819} C_VEL
LIN {X 0,Y 237.325,Z 558.558,A -85,B 0,C 180,E1 -20068.727,E2 -20068.727} C_VEL
LIN {X 0,Y 233.818,Z 567.506,A -85,B 0,C 180,E1 -20072.153,E2 -20072.153} C_VEL
LIN {X 0,Y 231.324,Z 574.142,A -85,B 0,C 180,E1 -20075.229,E2 -20075.229} C_VEL
LIN {X 0,Y 228.975,Z 580.458,A -85,B 0,C 180,E1 -20078.827,E2 -20078.827} C_VEL
LIN {X 0,Y 227.342,Z 585.503,A -85,B 0,C 180,E1 -20082.497,E2 -20082.497} C_VEL
LIN {X 0,Y 226.184,Z 589.46,A -85,B 0,C 180,E1 -20086.238,E2 -20086.238} C_VEL
LIN {X 0,Y 225.501,Z 592.263,A -85,B 0,C 180,E1 -20090.048,E2 -20090.048} C_VEL
LIN {X 0,Y 225.179,Z 593.961,A -85,B 0,C 180,E1 -20093.937,E2 -20093.937} C_VEL
LIN {X 0,Y 225.201,Z 594.577,A -85,B 0,C 180,E1 -20097.911,E2 -20097.911} C_VEL
LIN {X 0,Y 225.552,Z 593.949,A -85,B 0,C 180,E1 -20101.984,E2 -20101.984} C_VEL
LIN {X 0,Y 226.44,Z 592,A -85,B 0,C 180,E1 -20106.2,E2 -20106.2} C_VEL
LIN {X 0,Y 227.967,Z 588.768,A -85,B 0,C 180,E1 -20110.345,E2 -20110.345} C_VEL
LIN {X 0,Y 230.256,Z 584,A -85,B 0,C 180,E1 -20114.588,E2 -20114.588} C_VEL
LIN {X 0,Y 233.26,Z 578.146,A -85,B 0,C 180,E1 -20118.483,E2 -20118.483} C_VEL
LIN {X 0,Y 236.884,Z 571.265,A -85,B 0,C 180,E1 -20122.022,E2 -20122.022} C_VEL
LIN {X 0,Y 241.156,Z 563.223,A -85,B 0,C 180,E1 -20125.345,E2 -20125.345} C_VEL
LIN {X 0,Y 245.73,Z 554.488,A -85,B 0,C 180,E1 -20128.304,E2 -20128.304} C_VEL
LIN {X 0,Y 251.353,Z 543.262,A -85,B 0,C 180,E1 -20131.382,E2 -20131.382} C_VEL
LIN {X 0,Y 256.955,Z 531.185,A -85,B 0,C 180,E1 -20134.048,E2 -20134.048} C_VEL
LIN {X 0,Y 262.369,Z 518.525,A -85,B 0,C 180,E1 -20136.309,E2 -20136.309} C_VEL
LIN {X 0,Y 267.393,Z 505.46,A -85,B 0,C 180,E1 -20138.232,E2 -20138.232} C_VEL
LIN {X 0,Y 272.123,Z 491.713,A -85,B 0,C 180,E1 -20139.893,E2 -20139.893} C_VEL
LIN {X 0,Y 276.726,Z 476.39,A -85,B 0,C 180,E1 -20141.371,E2 -20141.371} C_VEL
LIN {X 0,Y 280.771,Z 460.008,A -85,B 0,C 180,E1 -20142.607,E2 -20142.607} C_VEL
LIN {X 0,Y 283.787,Z 444.455,A -85,B 0,C 180,E1 -20143.505,E2 -20143.505} C_VEL
LIN {X 0,Y 286.252,Z 427.923,A -85,B 0,C 180,E1 -20144.191,E2 -20144.191} C_VEL
LIN {X 0,Y 288.163,Z 407.195,A -85,B 0,C 180,E1 -20144.774,E2 -20144.774} C_VEL
LIN {X 0,Y 295.135,Z 314.957,A -85,B 0,C 180,E1 -20147.054,E2 -20147.054} C_VEL
LIN {X 0,Y 290.049,Z 305.49,A -85,B 0,C 180,E1 -20149.169,E2 -20149.169} C_VEL
LIN {X 0,Y 284.61,Z 296.099,A -85,B 0,C 180,E1 -20151.712,E2 -20151.712} C_VEL
LIN {X 0,Y 282.346,Z 292.557,A -85,B 0,C 180,E1 -20152.878,E2 -20152.878} C_VEL
LIN {X 0,Y 280.317,Z 290.446,A -85,B 0,C 180,E1 -20153.922,E2 -20153.922} C_VEL
LIN {X 0,Y 276.754,Z 288.791,A -85,B 0,C 180,E1 -20155.794,E2 -20155.794} C_VEL
LIN {X 0,Y 272.858,Z 287.224,A -85,B 0,C 180,E1 -20158.143,E2 -20158.143} C_VEL
LIN {X 0,Y 271.79,Z 286.191,A -85,B 0,C 180,E1 -20158.923,E2 -20158.923} C_VEL
LIN {X 0,Y 269.455,Z 282.376,A -85,B 0,C 180,E1 -20161.013,E2 -20161.013} C_VEL
LIN {X 0,Y 267.345,Z 279.22,A -85,B 0,C 180,E1 -20163.256,E2 -20163.256} C_VEL
LIN {X 0,Y 266.737,Z 278.379,A -85,B 0,C 180,E1 -20164.028,E2 -20164.028} C_VEL
LIN {X 0,Y 264.593,Z 276.487,A -85,B 0,C 180,E1 -20167.265,E2 -20167.265} C_VEL
LIN {X 0,Y 263.65,Z 273.567,A -85,B 0,C 180,E1 -20170.754,E2 -20170.754} C_VEL
LIN {X 0,Y 263.518,Z 273.362,A -85,B 0,C 180,E1 -20173.888,E2 -20173.888} C_VEL
LIN {X 0,Y 265.377,Z 277.679,A -85,B 0,C 180,E1 -20179.811,E2 -20179.811} C_VEL
LIN {X 0,Y 266.719,Z 278.777,A -85,B 0,C 180,E1 -20181.648,E2 -20181.648} C_VEL
LIN {X 0,Y 268.818,Z 282.204,A -85,B 0,C 180,E1 -20184.076,E2 -20184.076} C_VEL
LIN {X 0,Y 270.064,Z 283.65,A -85,B 0,C 180,E1 -20185.235,E2 -20185.235} C_VEL
LIN {X 0,Y 273.436,Z 288.734,A -85,B 0,C 180,E1 -20187.984,E2 -20187.984} C_VEL
LIN {X 0,Y 276.506,Z 293.872,A -85,B 0,C 180,E1 -20190.097,E2 -20190.097} C_VEL
LIN {X 0,Y 280.226,Z 300.462,A -85,B 0,C 180,E1 -20192.337,E2 -20192.337} C_VEL
LIN {X 0,Y 285.156,Z 310.387,A -85,B 0,C 180,E1 -20194.965,E2 -20194.965} C_VEL
LIN {X 0,Y 289.974,Z 321.084,A -85,B 0,C 180,E1 -20197.249,E2 -20197.249} C_VEL
LIN {X 0,Y 290.86,Z 323.173,A -85,B 0,C 180,E1 -20197.642,E2 -20197.642} C_VEL
LIN {X 0,Y 282.138,Z 432.479,A -85,B 0,C 180,E1 -20200.371,E2 -20200.371} C_VEL
LIN {X 0,Y 279.502,Z 450.423,A -85,B 0,C 180,E1 -20201.034,E2 -20201.034} C_VEL
LIN {X 0,Y 276.641,Z 464.313,A -85,B 0,C 180,E1 -20201.734,E2 -20201.734} C_VEL
LIN {X 0,Y 272.767,Z 479.883,A -85,B 0,C 180,E1 -20202.752,E2 -20202.752} C_VEL
LIN {X 0,Y 268.535,Z 494.344,A -85,B 0,C 180,E1 -20203.97,E2 -20203.97} C_VEL
LIN {X 0,Y 263.391,Z 509.19,A -85,B 0,C 180,E1 -20205.54,E2 -20205.54} C_VEL
LIN {X 0,Y 257.963,Z 522.991,A -85,B 0,C 180,E1 -20207.357,E2 -20207.357} C_VEL
LIN {X 0,Y 252.054,Z 536.625,A -85,B 0,C 180,E1 -20209.589,E2 -20209.589} C_VEL
LIN {X 0,Y 246.152,Z 549.166,A -85,B 0,C 180,E1 -20212.132,E2 -20212.132} C_VEL
LIN {X 0,Y 240.677,Z 560.108,A -85,B 0,C 180,E1 -20214.848,E2 -20214.848} C_VEL
LIN {X 0,Y 235.333,Z 570.307,A -85,B 0,C 180,E1 -20217.99,E2 -20217.99} C_VEL
LIN {X 0,Y 230.66,Z 579.062,A -85,B 0,C 180,E1 -20221.323,E2 -20221.323} C_VEL
LIN {X 0,Y 226.374,Z 587.274,A -85,B 0,C 180,E1 -20225.222,E2 -20225.222} C_VEL
LIN {X 0,Y 223.38,Z 593.298,A -85,B 0,C 180,E1 -20228.789,E2 -20228.789} C_VEL
LIN {X 0,Y 220.731,Z 599.177,A -85,B 0,C 180,E1 -20233.349,E2 -20233.349} C_VEL
LIN {X 0,Y 219.338,Z 602.647,A -85,B 0,C 180,E1 -20237.039,E2 -20237.039} C_VEL
LIN {X 0,Y 218.668,Z 605.209,A -85,B 0,C 180,E1 -20240.753,E2 -20240.753} C_VEL
LIN {X 0,Y 218.479,Z 607.042,A -85,B 0,C 180,E1 -20245.709,E2 -20245.709} C_VEL
LIN {X 0,Y 218.549,Z 607.304,A -85,B 0,C 180,E1 -20248.158,E2 -20248.158} C_VEL
LIN {X 0,Y 218.647,Z 607.183,A -85,B 0,C 180,E1 -20250.001,E2 -20250.001} C_VEL
LIN {X 0,Y 218.5,Z 606.249,A -85,B 0,C 180,E1 -20253.689,E2 -20253.689} C_VEL
LIN {X 0,Y 218.548,Z 605.44,A -85,B 0,C 180,E1 -20255.537,E2 -20255.537} C_VEL
LIN {X 0,Y 218.671,Z 602.927,A -85,B 0,C 180,E1 -20259.248,E2 -20259.248} C_VEL
LIN {X 0,Y 219.331,Z 599.431,A -85,B 0,C 180,E1 -20262.962,E2 -20262.962} C_VEL
LIN {X 0,Y 220.955,Z 593.714,A -85,B 0,C 180,E1 -20267.404,E2 -20267.404} C_VEL
LIN {X 0,Y 223.056,Z 587.244,A -85,B 0,C 180,E1 -20271.244,E2 -20271.244} C_VEL
LIN {X 0,Y 225.879,Z 579.712,A -85,B 0,C 180,E1 -20274.837,E2 -20274.837} C_VEL
LIN {X 0,Y 229.464,Z 570.687,A -85,B 0,C 180,E1 -20278.342,E2 -20278.342} C_VEL
LIN {X 0,Y 233.321,Z 561.388,A -85,B 0,C 180,E1 -20281.305,E2 -20281.305} C_VEL
LIN {X 0,Y 237.531,Z 550.389,A -85,B 0,C 180,E1 -20284.206,E2 -20284.206} C_VEL
LIN {X 0,Y 242.487,Z 537.475,A -85,B 0,C 180,E1 -20286.97,E2 -20286.97} C_VEL
LIN {X 0,Y 246.769,Z 525.598,A -85,B 0,C 180,E1 -20289.059,E2 -20289.059} C_VEL
LIN {X 0,Y 251.136,Z 512.367,A -85,B 0,C 180,E1 -20290.99,E2 -20290.99} C_VEL
LIN {X 0,Y 255.309,Z 498.056,A -85,B 0,C 180,E1 -20292.677,E2 -20292.677} C_VEL
LIN {X 0,Y 259.253,Z 482.595,A -85,B 0,C 180,E1 -20294.135,E2 -20294.135} C_VEL
LIN {X 0,Y 262.607,Z 466.772,A -85,B 0,C 180,E1 -20295.306,E2 -20295.306} C_VEL
LIN {X 0,Y 265.365,Z 450.962,A -85,B 0,C 180,E1 -20296.181,E2 -20296.181} C_VEL
LIN {X 0,Y 267.606,Z 433.572,A -85,B 0,C 180,E1 -20296.852,E2 -20296.852} C_VEL
LIN {X 0,Y 275.236,Z 316.331,A -85,B 0,C 180,E1 -20299.852,E2 -20299.852} C_VEL
LIN {X 0,Y 268.359,Z 301.752,A -85,B 0,C 180,E1 -20301.933,E2 -20301.933} C_VEL
LIN {X 0,Y 259.585,Z 285.163,A -85,B 0,C 180,E1 -20304.759,E2 -20304.759} C_VEL
LIN {X 0,Y 252.695,Z 273.265,A -85,B 0,C 180,E1 -20307.167,E2 -20307.167} C_VEL
LIN {X 0,Y 247.942,Z 265.776,A -85,B 0,C 180,E1 -20308.923,E2 -20308.923} C_VEL
LIN {X 0,Y 243.105,Z 259.2,A -85,B 0,C 180,E1 -20310.794,E2 -20310.794} C_VEL
LIN {X 0,Y 239.837,Z 254.898,A -85,B 0,C 180,E1 -20312.122,E2 -20312.122} C_VEL
LIN {X 0,Y 236.695,Z 250.707,A -85,B 0,C 180,E1 -20313.474,E2 -20313.474} C_VEL
LIN {X 0,Y 233.927,Z 247.058,A -85,B 0,C 180,E1 -20314.737,E2 -20314.737} C_VEL
LIN {X 0,Y 232.482,Z 245.418,A -85,B 0,C 180,E1 -20315.409,E2 -20315.409} C_VEL
LIN {X 0,Y 230.061,Z 242.212,A -85,B 0,C 180,E1 -20316.601,E2 -20316.601} C_VEL
LIN {X 0,Y 229.402,Z 241.286,A -85,B 0,C 180,E1 -20316.938,E2 -20316.938} C_VEL
LIN {X 0,Y 226.78,Z 238.835,A -85,B 0,C 180,E1 -20318.228,E2 -20318.228} C_VEL
LIN {X 0,Y 225.096,Z 235.867,A -85,B 0,C 180,E1 -20319.197,E2 -20319.197} C_VEL
LIN {X 0,Y 222.521,Z 233.978,A -85,B 0,C 180,E1 -20320.573,E2 -20320.573} C_VEL
LIN {X 0,Y 221.214,Z 231.625,A -85,B 0,C 180,E1 -20321.416,E2 -20321.416} C_VEL
LIN {X 0,Y 220.893,Z 230.242,A -85,B 0,C 180,E1 -20321.714,E2 -20321.714} C_VEL
LIN {X 0,Y 220.967,Z 230.259,A -85,B 0,C 180,E1 -20325.259,E2 -20325.259} C_VEL
LIN {X 0,Y 221.186,Z 230.218,A -85,B 0,C 180,E1 -20330.859,E2 -20330.859} C_VEL
LIN {X 0,Y 221.25,Z 230.238,A -85,B 0,C 180,E1 -20332.7,E2 -20332.7} C_VEL
LIN {X 0,Y 221.509,Z 230.148,A -85,B 0,C 180,E1 -20338.182,E2 -20338.182} C_VEL
LIN {X 0,Y 221.511,Z 230.207,A -85,B 0,C 180,E1 -20341.818,E2 -20341.818} C_VEL
LIN {X 0,Y 221.259,Z 230.223,A -85,B 0,C 180,E1 -20347.299,E2 -20347.299} C_VEL
LIN {X 0,Y 221.067,Z 230.23,A -85,B 0,C 180,E1 -20350.996,E2 -20350.996} C_VEL
LIN {X 0,Y 220.996,Z 230.264,A -85,B 0,C 180,E1 -20354.739,E2 -20354.739} C_VEL
LIN {X 0,Y 220.922,Z 230.244,A -85,B 0,C 180,E1 -20358.549,E2 -20358.549} C_VEL
LIN {X 0,Y 220.896,Z 230.28,A -85,B 0,C 180,E1 -20362.683,E2 -20362.683} C_VEL
LIN {X 0,Y 220.887,Z 230.261,A -85,B 0,C 180,E1 -20367.016,E2 -20367.016} C_VEL
LIN {X 0,Y 220.863,Z 230.263,A -85,B 0,C 180,E1 -20370.778,E2 -20370.778} C_VEL
LIN {X 0,Y 220.801,Z 230.294,A -85,B 0,C 180,E1 -20374.955,E2 -20374.955} C_VEL
LIN {X 0,Y 220.806,Z 230.274,A -85,B 0,C 180,E1 -20379.537,E2 -20379.537} C_VEL
LIN {X 0,Y 220.807,Z 230.304,A -85,B 0,C 180,E1 -20384.796,E2 -20384.796} C_VEL
LIN {X 0,Y 221.527,Z 232.671,A -85,B 0,C 180,E1 -20385.352,E2 -20385.352} C_VEL
LIN {X 0,Y 223.27,Z 234.891,A -85,B 0,C 180,E1 -20386.384,E2 -20386.384} C_VEL
LIN {X 0,Y 225.297,Z 236.267,A -85,B 0,C 180,E1 -20387.439,E2 -20387.439} C_VEL
LIN {X 0,Y 227.151,Z 239.406,A -85,B 0,C 180,E1 -20388.485,E2 -20388.485} C_VEL
LIN {X 0,Y 229.797,Z 241.878,A -85,B 0,C 180,E1 -20389.795,E2 -20389.795} C_VEL
LIN {X 0,Y 232.345,Z 245.426,A -85,B 0,C 180,E1 -20391.064,E2 -20391.064} C_VEL
LIN {X 0,Y 233.921,Z 247.074,A -85,B 0,C 180,E1 -20391.781,E2 -20391.781} C_VEL
LIN {X 0,Y 236.603,Z 250.643,A -85,B 0,C 180,E1 -20392.995,E2 -20392.995} C_VEL
LIN {X 0,Y 238.357,Z 252.965,A -85,B 0,C 180,E1 -20393.766,E2 -20393.766} C_VEL
LIN {X 0,Y 241.832,Z 257.489,A -85,B 0,C 180,E1 -20395.217,E2 -20395.217} C_VEL
LIN {X 0,Y 246.065,Z 263.178,A -85,B 0,C 180,E1 -20396.882,E2 -20396.882} C_VEL
LIN {X 0,Y 253.029,Z 272.963,A -85,B 0,C 180,E1 -20399.433,E2 -20399.433} C_VEL
LIN {X 0,Y 263.184,Z 288.731,A -85,B 0,C 180,E1 -20402.811,E2 -20402.811} C_VEL
LIN {X 0,Y 271.916,Z 303.66,A -85,B 0,C 180,E1 -20405.452,E2 -20405.452} C_VEL
LIN {X 0,Y 275.334,Z 309.962,A -85,B 0,C 180,E1 -20406.433,E2 -20406.433} C_VEL
LIN {X 0,Y 268.058,Z 421.22,A -85,B 0,C 180,E1 -20409.271,E2 -20409.271} C_VEL
LIN {X 0,Y 266.009,Z 438.547,A -85,B 0,C 180,E1 -20409.962,E2 -20409.962} C_VEL
LIN {X 0,Y 263.336,Z 455.148,A -85,B 0,C 180,E1 -20410.917,E2 -20410.917} C_VEL
LIN {X 0,Y 260.147,Z 470.775,A -85,B 0,C 180,E1 -20412.103,E2 -20412.103} C_VEL
LIN {X 0,Y 256.413,Z 486.204,A -85,B 0,C 180,E1 -20413.599,E2 -20413.599} C_VEL
LIN {X 0,Y 252.376,Z 500.331,A -85,B 0,C 180,E1 -20415.279,E2 -20415.279} C_VEL
LIN {X 0,Y 248.004,Z 514.062,A -85,B 0,C 180,E1 -20417.313,E2 -20417.313} C_VEL
LIN {X 0,Y 243.48,Z 526.786,A -85,B 0,C 180,E1 -20419.603,E2 -20419.603} C_VEL
LIN {X 0,Y 238.71,Z 539.414,A -85,B 0,C 180,E1 -20422.386,E2 -20422.386} C_VEL
LIN {X 0,Y 234.356,Z 550.178,A -85,B 0,C 180,E1 -20425.269,E2 -20425.269} C_VEL
LIN {X 0,Y 230.532,Z 559.4,A -85,B 0,C 180,E1 -20428.253,E2 -20428.253} C_VEL
LIN {X 0,Y 226.918,Z 568.235,A -85,B 0,C 180,E1 -20431.774,E2 -20431.774} C_VEL
LIN {X 0,Y 223.991,Z 575.607,A -85,B 0,C 180,E1 -20435.401,E2 -20435.401} C_VEL
LIN {X 0,Y 221.674,Z 581.71,A -85,B 0,C 180,E1 -20439.12,E2 -20439.12} C_VEL
LIN {X 0,Y 220.07,Z 586.557,A -85,B 0,C 180,E1 -20442.917,E2 -20442.917} C_VEL
LIN {X 0,Y 218.953,Z 590.252,A -85,B 0,C 180,E1 -20446.79,E2 -20446.79} C_VEL
LIN {X 0,Y 218.283,Z 593.005,A -85,B 0,C 180,E1 -20450.981,E2 -20450.981} C_VEL
LIN {X 0,Y 218.047,Z 594.379,A -85,B 0,C 180,E1 -20454.771,E2 -20454.771} C_VEL
LIN {X 0,Y 218.167,Z 594.73,A -85,B 0,C 180,E1 -20458.894,E2 -20458.894} C_VEL
LIN {X 0,Y 218.671,Z 593.828,A -85,B 0,C 180,E1 -20463.319,E2 -20463.319} C_VEL
LIN {X 0,Y 219.701,Z 591.767,A -85,B 0,C 180,E1 -20467.429,E2 -20467.429} C_VEL
LIN {X 0,Y 221.526,Z 588.196,A -85,B 0,C 180,E1 -20471.776,E2 -20471.776} C_VEL
LIN {X 0,Y 224.181,Z 583.109,A -85,B 0,C 180,E1 -20476.139,E2 -20476.139} C_VEL
LIN {X 0,Y 226.894,Z 578.176,A -85,B 0,C 180,E1 -20479.423,E2 -20479.423} C_VEL
LIN {X 0,Y 230.797,Z 571.22,A -85,B 0,C 180,E1 -20483.065,E2 -20483.065} C_VEL
LIN {X 0,Y 235.613,Z 562.658,A -85,B 0,C 180,E1 -20486.635,E2 -20486.635} C_VEL
LIN {X 0,Y 241.139,Z 552.531,A -85,B 0,C 180,E1 -20489.999,E2 -20489.999} C_VEL
LIN {X 0,Y 246.703,Z 541.754,A -85,B 0,C 180,E1 -20492.884,E2 -20492.884} C_VEL
LIN {X 0,Y 252.01,Z 530.874,A -85,B 0,C 180,E1 -20495.272,E2 -20495.272} C_VEL
LIN {X 0,Y 257.624,Z 518.186,A -85,B 0,C 180,E1 -20497.547,E2 -20497.547} C_VEL
LIN {X 0,Y 263.056,Z 504.525,A -85,B 0,C 180,E1 -20499.542,E2 -20499.542} C_VEL
LIN {X 0,Y 268.323,Z 489.48,A -85,B 0,C 180,E1 -20501.307,E2 -20501.307} C_VEL
LIN {X 0,Y 272.784,Z 474.683,A -85,B 0,C 180,E1 -20502.691,E2 -20502.691} C_VEL
LIN {X 0,Y 276.657,Z 459.253,A -85,B 0,C 180,E1 -20503.842,E2 -20503.842} C_VEL
LIN {X 0,Y 280.042,Z 442.212,A -85,B 0,C 180,E1 -20504.798,E2 -20504.798} C_VEL
LIN {X 0,Y 282.466,Z 425.718,A -85,B 0,C 180,E1 -20505.437,E2 -20505.437} C_VEL
LIN {X 0,Y 284.691,Z 400.233,A -85,B 0,C 180,E1 -20506.121,E2 -20506.121} C_VEL
LIN {X 0,Y 291.082,Z 318.371,A -85,B 0,C 180,E1 -20508.158,E2 -20508.158} C_VEL
LIN {X 0,Y 286.61,Z 309.839,A -85,B 0,C 180,E1 -20510.159,E2 -20510.159} C_VEL
LIN {X 0,Y 281.896,Z 301.541,A -85,B 0,C 180,E1 -20512.502,E2 -20512.502} C_VEL
LIN {X 0,Y 277.497,Z 294.546,A -85,B 0,C 180,E1 -20514.981,E2 -20514.981} C_VEL
LIN {X 0,Y 274.83,Z 290.44,A -85,B 0,C 180,E1 -20516.699,E2 -20516.699} C_VEL
LIN {X 0,Y 272.693,Z 287.245,A -85,B 0,C 180,E1 -20518.241,E2 -20518.241} C_VEL
LIN {X 0,Y 271.79,Z 286.191,A -85,B 0,C 180,E1 -20518.923,E2 -20518.923} C_VEL
LIN {X 0,Y 270.282,Z 284.921,A -85,B 0,C 180,E1 -20520.102,E2 -20520.102} C_VEL
LIN {X 0,Y 267.803,Z 284.624,A -85,B 0,C 180,E1 -20522.144,E2 -20522.144} C_VEL
LIN {X 0,Y 265.275,Z 284.974,A -85,B 0,C 180,E1 -20524.675,E2 -20524.675} C_VEL
LIN {X 0,Y 264.626,Z 284.733,A -85,B 0,C 180,E1 -20525.529,E2 -20525.529} C_VEL
LIN {X 0,Y 262.904,Z 281.869,A -85,B 0,C 180,E1 -20529.364,E2 -20529.364} C_VEL
LIN {X 0,Y 262.628,Z 280.494,A -85,B 0,C 180,E1 -20531.234,E2 -20531.234} C_VEL
LIN {X 0,Y 262.584,Z 280.614,A -85,B 0,C 180,E1 -20534.218,E2 -20534.218} C_VEL
LIN {X 0,Y 264.157,Z 284.466,A -85,B 0,C 180,E1 -20539.393,E2 -20539.393} C_VEL
LIN {X 0,Y 265.526,Z 285.731,A -85,B 0,C 180,E1 -20541.374,E2 -20541.374} C_VEL
LIN {X 0,Y 267.683,Z 289.21,A -85,B 0,C 180,E1 -20543.936,E2 -20543.936} C_VEL
LIN {X 0,Y 268.698,Z 290.525,A -85,B 0,C 180,E1 -20544.92,E2 -20544.92} C_VEL
LIN {X 0,Y 271.897,Z 295.462,A -85,B 0,C 180,E1 -20547.623,E2 -20547.623} C_VEL
LIN {X 0,Y 274.696,Z 300.428,A -85,B 0,C 180,E1 -20549.639,E2 -20549.639} C_VEL
LIN {X 0,Y 278.044,Z 306.623,A -85,B 0,C 180,E1 -20551.76,E2 -20551.76} C_VEL
LIN {X 0,Y 282.514,Z 316.067,A -85,B 0,C 180,E1 -20554.28,E2 -20554.28} C_VEL
LIN {X 0,Y 286.773,Z 325.86,A -85,B 0,C 180,E1 -20556.408,E2 -20556.408} C_VEL
LIN {X 0,Y 286.988,Z 326.88,A -85,B 0,C 180,E1 -20556.538,E2 -20556.538} C_VEL
LIN {X 0,Y 278.205,Z 432.141,A -85,B 0,C 180,E1 -20559.15,E2 -20559.15} C_VEL
LIN {X 0,Y 275.55,Z 449.864,A -85,B 0,C 180,E1 -20559.802,E2 -20559.802} C_VEL
LIN {X 0,Y 272.345,Z 465.03,A -85,B 0,C 180,E1 -20560.568,E2 -20560.568} C_VEL
LIN {X 0,Y 268.62,Z 479.381,A -85,B 0,C 180,E1 -20561.504,E2 -20561.504} C_VEL
LIN {X 0,Y 264.238,Z 493.829,A -85,B 0,C 180,E1 -20562.716,E2 -20562.716} C_VEL
LIN {X 0,Y 258.942,Z 508.667,A -85,B 0,C 180,E1 -20564.289,E2 -20564.289} C_VEL
LIN {X 0,Y 253.848,Z 521.277,A -85,B 0,C 180,E1 -20565.926,E2 -20565.926} C_VEL
LIN {X 0,Y 248.583,Z 533.293,A -85,B 0,C 180,E1 -20567.821,E2 -20567.821} C_VEL
LIN {X 0,Y 242.255,Z 546.267,A -85,B 0,C 180,E1 -20570.341,E2 -20570.341} C_VEL
LIN {X 0,Y 236.501,Z 557.294,A -85,B 0,C 180,E1 -20573.005,E2 -20573.005} C_VEL
LIN {X 0,Y 230.69,Z 568.059,A -85,B 0,C 180,E1 -20576.222,E2 -20576.222} C_VEL
LIN {X 0,Y 225.558,Z 577.18,A -85,B 0,C 180,E1 -20579.582,E2 -20579.582} C_VEL
LIN {X 0,Y 220.757,Z 585.707,A -85,B 0,C 180,E1 -20583.533,E2 -20583.533} C_VEL
LIN {X 0,Y 217.402,Z 591.883,A -85,B 0,C 180,E1 -20587.175,E2 -20587.175} C_VEL
LIN {X 0,Y 214.832,Z 596.957,A -85,B 0,C 180,E1 -20590.906,E2 -20590.906} C_VEL
LIN {X 0,Y 213.021,Z 600.96,A -85,B 0,C 180,E1 -20594.697,E2 -20594.697} C_VEL
LIN {X 0,Y 211.885,Z 603.919,A -85,B 0,C 180,E1 -20598.521,E2 -20598.521} C_VEL
LIN {X 0,Y 211.414,Z 605.914,A -85,B 0,C 180,E1 -20602.359,E2 -20602.359} C_VEL
LIN {X 0,Y 211.375,Z 606.916,A -85,B 0,C 180,E1 -20606.188,E2 -20606.188} C_VEL
LIN {X 0,Y 211.563,Z 606.966,A -85,B 0,C 180,E1 -20610.001,E2 -20610.001} C_VEL
LIN {X 0,Y 211.445,Z 605.767,A -85,B 0,C 180,E1 -20614.339,E2 -20614.339} C_VEL
LIN {X 0,Y 211.433,Z 604.017,A -85,B 0,C 180,E1 -20617.641,E2 -20617.641} C_VEL
LIN {X 0,Y 211.876,Z 600.966,A -85,B 0,C 180,E1 -20621.48,E2 -20621.48} C_VEL
LIN {X 0,Y 212.949,Z 596.887,A -85,B 0,C 180,E1 -20625.309,E2 -20625.309} C_VEL
LIN {X 0,Y 214.607,Z 591.554,A -85,B 0,C 180,E1 -20629.116,E2 -20629.116} C_VEL
LIN {X 0,Y 217.013,Z 585.024,A -85,B 0,C 180,E1 -20632.869,E2 -20632.869} C_VEL
LIN {X 0,Y 220.365,Z 576.621,A -85,B 0,C 180,E1 -20636.749,E2 -20636.749} C_VEL
LIN {X 0,Y 224.734,Z 566.283,A -85,B 0,C 180,E1 -20640.543,E2 -20640.543} C_VEL
LIN {X 0,Y 228.417,Z 557.704,A -85,B 0,C 180,E1 -20643.102,E2 -20643.102} C_VEL
LIN {X 0,Y 232.283,Z 547.954,A -85,B 0,C 180,E1 -20645.622,E2 -20645.622} C_VEL
LIN {X 0,Y 237.513,Z 534.612,A -85,B 0,C 180,E1 -20648.418,E2 -20648.418} C_VEL
LIN {X 0,Y 242.432,Z 521,A -85,B 0,C 180,E1 -20650.713,E2 -20650.713} C_VEL
LIN {X 0,Y 246.747,Z 507.858,A -85,B 0,C 180,E1 -20652.516,E2 -20652.516} C_VEL
LIN {X 0,Y 251.02,Z 493.309,A -85,B 0,C 180,E1 -20654.142,E2 -20654.142} C_VEL
LIN {X 0,Y 254.861,Z 477.926,A -85,B 0,C 180,E1 -20655.522,E2 -20655.522} C_VEL
LIN {X 0,Y 258.074,Z 462.178,A -85,B 0,C 180,E1 -20656.616,E2 -20656.616} C_VEL
LIN {X 0,Y 260.848,Z 445.436,A -85,B 0,C 180,E1 -20657.449,E2 -20657.449} C_VEL
LIN {X 0,Y 262.696,Z 429.38,A -85,B 0,C 180,E1 -20658.007,E2 -20658.007} C_VEL
LIN {X 0,Y 270.064,Z 318.731,A -85,B 0,C 180,E1 -20660.861,E2 -20660.861} C_VEL
LIN {X 0,Y 262.879,Z 303.588,A -85,B 0,C 180,E1 -20663.14,E2 -20663.14} C_VEL
LIN {X 0,Y 254.368,Z 287.529,A -85,B 0,C 180,E1 -20666.03,E2 -20666.03} C_VEL
LIN {X 0,Y 248.995,Z 278.202,A -85,B 0,C 180,E1 -20667.987,E2 -20667.987} C_VEL
LIN {X 0,Y 244.361,Z 270.699,A -85,B 0,C 180,E1 -20669.782,E2 -20669.782} C_VEL
LIN {X 0,Y 237.098,Z 260.911,A -85,B 0,C 180,E1 -20672.742,E2 -20672.742} C_VEL
LIN {X 0,Y 233.869,Z 256.627,A -85,B 0,C 180,E1 -20674.181,E2 -20674.181} C_VEL
LIN {X 0,Y 230.43,Z 252.056,A -85,B 0,C 180,E1 -20675.821,E2 -20675.821} C_VEL
LIN {X 0,Y 227.67,Z 248.55,A -85,B 0,C 180,E1 -20677.195,E2 -20677.195} C_VEL
LIN {X 0,Y 226.497,Z 247.248,A -85,B 0,C 180,E1 -20677.785,E2 -20677.785} C_VEL
LIN {X 0,Y 223.841,Z 244.176,A -85,B 0,C 180,E1 -20679.196,E2 -20679.196} C_VEL
LIN {X 0,Y 222.807,Z 242.331,A -85,B 0,C 180,E1 -20679.818,E2 -20679.818} C_VEL
LIN {X 0,Y 220.145,Z 240.04,A -85,B 0,C 180,E1 -20681.323,E2 -20681.323} C_VEL
LIN {X 0,Y 218.574,Z 237.085,A -85,B 0,C 180,E1 -20682.386,E2 -20682.386} C_VEL
LIN {X 0,Y 215.5,Z 234.81,A -85,B 0,C 180,E1 -20684.271,E2 -20684.271} C_VEL
LIN {X 0,Y 214.251,Z 232.511,A -85,B 0,C 180,E1 -20685.212,E2 -20685.212} C_VEL
LIN {X 0,Y 213.919,Z 231.127,A -85,B 0,C 180,E1 -20685.614,E2 -20685.614} C_VEL
LIN {X 0,Y 214.125,Z 231.09,A -85,B 0,C 180,E1 -20690.555,E2 -20690.555} C_VEL
LIN {X 0,Y 214.092,Z 231.095,A -85,B 0,C 180,E1 -20694.348,E2 -20694.348} C_VEL
LIN {X 0,Y 214.442,Z 231.027,A -85,B 0,C 180,E1 -20698.122,E2 -20698.122} C_VEL
LIN {X 0,Y 214.546,Z 231.045,A -85,B 0,C 180,E1 -20700,E2 -20700} C_VEL
LIN {X 0,Y 214.444,Z 231.087,A -85,B 0,C 180,E1 -20701.878,E2 -20701.878} C_VEL
LIN {X 0,Y 214.198,Z 231.106,A -85,B 0,C 180,E1 -20707.541,E2 -20707.541} C_VEL
LIN {X 0,Y 213.999,Z 231.107,A -85,B 0,C 180,E1 -20711.364,E2 -20711.364} C_VEL
LIN {X 0,Y 213.935,Z 231.147,A -85,B 0,C 180,E1 -20715.237,E2 -20715.237} C_VEL
LIN {X 0,Y 213.839,Z 231.126,A -85,B 0,C 180,E1 -20719.187,E2 -20719.187} C_VEL
LIN {X 0,Y 213.848,Z 231.148,A -85,B 0,C 180,E1 -20723.227,E2 -20723.227} C_VEL
LIN {X 0,Y 213.829,Z 231.145,A -85,B 0,C 180,E1 -20727.45,E2 -20727.45} C_VEL
LIN {X 0,Y 213.777,Z 231.139,A -85,B 0,C 180,E1 -20731.736,E2 -20731.736} C_VEL
LIN {X 0,Y 213.744,Z 231.16,A -85,B 0,C 180,E1 -20736.288,E2 -20736.288} C_VEL
LIN {X 0,Y 213.718,Z 231.186,A -85,B 0,C 180,E1 -20740.857,E2 -20740.857} C_VEL
LIN {X 0,Y 214.434,Z 233.482,A -85,B 0,C 180,E1 -20741.503,E2 -20741.503} C_VEL
LIN {X 0,Y 216.239,Z 235.755,A -85,B 0,C 180,E1 -20742.754,E2 -20742.754} C_VEL
LIN {X 0,Y 218.542,Z 237.273,A -85,B 0,C 180,E1 -20744.141,E2 -20744.141} C_VEL
LIN {X 0,Y 220.069,Z 240.133,A -85,B 0,C 180,E1 -20745.174,E2 -20745.174} C_VEL
LIN {X 0,Y 222.551,Z 242.33,A -85,B 0,C 180,E1 -20746.579,E2 -20746.579} C_VEL
LIN {X 0,Y 225.734,Z 246.622,A -85,B 0,C 180,E1 -20748.349,E2 -20748.349} C_VEL
LIN {X 0,Y 227.443,Z 248.282,A -85,B 0,C 180,E1 -20749.213,E2 -20749.213} C_VEL
LIN {X 0,Y 230.208,Z 251.97,A -85,B 0,C 180,E1 -20750.613,E2 -20750.613} C_VEL
LIN {X 0,Y 231.471,Z 253.485,A -85,B 0,C 180,E1 -20751.217,E2 -20751.217} C_VEL
LIN {X 0,Y 235.447,Z 258.705,A -85,B 0,C 180,E1 -20753.042,E2 -20753.042} C_VEL
LIN {X 0,Y 241.911,Z 267.369,A -85,B 0,C 180,E1 -20755.776,E2 -20755.776} C_VEL
LIN {X 0,Y 249.448,Z 278.077,A -85,B 0,C 180,E1 -20758.658,E2 -20758.658} C_VEL
LIN {X 0,Y 259.367,Z 293.714,A -85,B 0,C 180,E1 -20762.081,E2 -20762.081} C_VEL
LIN {X 0,Y 268.354,Z 309.325,A -85,B 0,C 180,E1 -20764.887,E2 -20764.887} C_VEL
LIN {X 0,Y 270.216,Z 312.786,A -85,B 0,C 180,E1 -20765.444,E2 -20765.444} C_VEL
LIN {X 0,Y 262.871,Z 420.977,A -85,B 0,C 180,E1 -20768.225,E2 -20768.225} C_VEL
LIN {X 0,Y 260.888,Z 437.555,A -85,B 0,C 180,E1 -20768.881,E2 -20768.881} C_VEL
LIN {X 0,Y 258.238,Z 453.858,A -85,B 0,C 180,E1 -20769.8,E2 -20769.8} C_VEL
LIN {X 0,Y 254.979,Z 469.796,A -85,B 0,C 180,E1 -20770.999,E2 -20770.999} C_VEL
LIN {X 0,Y 251.165,Z 485.246,A -85,B 0,C 180,E1 -20772.483,E2 -20772.483} C_VEL
LIN {X 0,Y 246.708,Z 500.417,A -85,B 0,C 180,E1 -20774.298,E2 -20774.298} C_VEL
LIN {X 0,Y 242.178,Z 514.167,A -85,B 0,C 180,E1 -20776.362,E2 -20776.362} C_VEL
LIN {X 0,Y 237.936,Z 525.717,A -85,B 0,C 180,E1 -20778.449,E2 -20778.449} C_VEL
LIN {X 0,Y 233.562,Z 537.082,A -85,B 0,C 180,E1 -20780.91,E2 -20780.91} C_VEL
LIN {X 0,Y 228.937,Z 548.215,A -85,B 0,C 180,E1 -20783.832,E2 -20783.832} C_VEL
LIN {X 0,Y 224.316,Z 558.945,A -85,B 0,C 180,E1 -20787.305,E2 -20787.305} C_VEL
LIN {X 0,Y 220.464,Z 567.915,A -85,B 0,C 180,E1 -20790.913,E2 -20790.913} C_VEL
LIN {X 0,Y 217.371,Z 575.392,A -85,B 0,C 180,E1 -20794.636,E2 -20794.636} C_VEL
LIN {X 0,Y 214.886,Z 581.593,A -85,B 0,C 180,E1 -20798.463,E2 -20798.463} C_VEL
LIN {X 0,Y 213.16,Z 586.483,A -85,B 0,C 180,E1 -20802.374,E2 -20802.374} C_VEL
LIN {X 0,Y 212.04,Z 589.991,A -85,B 0,C 180,E1 -20806.015,E2 -20806.015} C_VEL
LIN {X 0,Y 211.366,Z 592.376,A -85,B 0,C 180,E1 -20809.42,E2 -20809.42} C_VEL
LIN {X 0,Y 210.997,Z 594.241,A -85,B 0,C 180,E1 -20813.559,E2 -20813.559} C_VEL
LIN {X 0,Y 210.954,Z 594.798,A -85,B 0,C 180,E1 -20815.906,E2 -20815.906} C_VEL
LIN {X 0,Y 211.147,Z 594.878,A -85,B 0,C 180,E1 -20820.071,E2 -20820.071} C_VEL
LIN {X 0,Y 211.759,Z 593.79,A -85,B 0,C 180,E1 -20824.346,E2 -20824.346} C_VEL
LIN {X 0,Y 213.091,Z 591.406,A -85,B 0,C 180,E1 -20828.802,E2 -20828.802} C_VEL
LIN {X 0,Y 215.186,Z 587.604,A -85,B 0,C 180,E1 -20833.302,E2 -20833.302} C_VEL
LIN {X 0,Y 218.27,Z 582.223,A -85,B 0,C 180,E1 -20837.778,E2 -20837.778} C_VEL
LIN {X 0,Y 221.441,Z 576.816,A -85,B 0,C 180,E1 -20841.217,E2 -20841.217} C_VEL
LIN {X 0,Y 225.632,Z 569.869,A -85,B 0,C 180,E1 -20844.786,E2 -20844.786} C_VEL
LIN {X 0,Y 230.937,Z 560.892,A -85,B 0,C 180,E1 -20848.44,E2 -20848.44} C_VEL
LIN {X 0,Y 237.094,Z 550.069,A -85,B 0,C 180,E1 -20851.906,E2 -20851.906} C_VEL
LIN {X 0,Y 242.875,Z 539.108,A -85,B 0,C 180,E1 -20854.722,E2 -20854.722} C_VEL
LIN {X 0,Y 248.561,Z 527.662,A -85,B 0,C 180,E1 -20857.103,E2 -20857.103} C_VEL
LIN {X 0,Y 254.388,Z 514.668,A -85,B 0,C 180,E1 -20859.327,E2 -20859.327} C_VEL
LIN {X 0,Y 259.829,Z 501.157,A -85,B 0,C 180,E1 -20861.206,E2 -20861.206} C_VEL
LIN {X 0,Y 264.218,Z 488.812,A -85,B 0,C 180,E1 -20862.597,E2 -20862.597} C_VEL
LIN {X 0,Y 268.822,Z 473.838,A -85,B 0,C 180,E1 -20863.985,E2 -20863.985} C_VEL
LIN {X 0,Y 272.717,Z 458.624,A -85,B 0,C 180,E1 -20865.102,E2 -20865.102} C_VEL
LIN {X 0,Y 276.013,Z 442.532,A -85,B 0,C 180,E1 -20865.995,E2 -20865.995} C_VEL
LIN {X 0,Y 278.526,Z 425.833,A -85,B 0,C 180,E1 -20866.645,E2 -20866.645} C_VEL
LIN {X 0,Y 281.037,Z 397.804,A -85,B 0,C 180,E1 -20867.386,E2 -20867.386} C_VEL
LIN {X 0,Y 287.259,Z 321.932,A -85,B 0,C 180,E1 -20869.264,E2 -20869.264} C_VEL
LIN {X 0,Y 282.751,Z 313.306,A -85,B 0,C 180,E1 -20871.423,E2 -20871.423} C_VEL
LIN {X 0,Y 278.428,Z 305.542,A -85,B 0,C 180,E1 -20873.767,E2 -20873.767} C_VEL
LIN {X 0,Y 273.54,Z 297.56,A -85,B 0,C 180,E1 -20876.851,E2 -20876.851} C_VEL
LIN {X 0,Y 271.03,Z 293.81,A -85,B 0,C 180,E1 -20878.718,E2 -20878.718} C_VEL
LIN {X 0,Y 268.479,Z 289.782,A -85,B 0,C 180,E1 -20880.968,E2 -20880.968} C_VEL
LIN {X 0,Y 265.931,Z 285.673,A -85,B 0,C 180,E1 -20883.815,E2 -20883.815} C_VEL
LIN {X 0,Y 264.626,Z 284.733,A -85,B 0,C 180,E1 -20885.529,E2 -20885.529} C_VEL
LIN {X 0,Y 263.515,Z 284.707,A -85,B 0,C 180,E1 -20887.223,E2 -20887.223} C_VEL
LIN {X 0,Y 261.68,Z 287.25,A -85,B 0,C 180,E1 -20891.499,E2 -20891.499} C_VEL
LIN {X 0,Y 261.568,Z 287.382,A -85,B 0,C 180,E1 -20892.367,E2 -20892.367} C_VEL
LIN {X 0,Y 261.621,Z 287.817,A -85,B 0,C 180,E1 -20894.272,E2 -20894.272} C_VEL
LIN {X 0,Y 263.331,Z 291.695,A -85,B 0,C 180,E1 -20899.628,E2 -20899.628} C_VEL
LIN {X 0,Y 264.335,Z 292.688,A -85,B 0,C 180,E1 -20901.093,E2 -20901.093} C_VEL
LIN {X 0,Y 266.604,Z 296.302,A -85,B 0,C 180,E1 -20903.852,E2 -20903.852} C_VEL
LIN {X 0,Y 267.508,Z 297.745,A -85,B 0,C 180,E1 -20904.775,E2 -20904.775} C_VEL
LIN {X 0,Y 270.267,Z 302.063,A -85,B 0,C 180,E1 -20907.175,E2 -20907.175} C_VEL
LIN {X 0,Y 272.621,Z 306.457,A -85,B 0,C 180,E1 -20908.978,E2 -20908.978} C_VEL
LIN {X 0,Y 275.93,Z 312.817,A -85,B 0,C 180,E1 -20911.189,E2 -20911.189} C_VEL
LIN {X 0,Y 280.131,Z 322.149,A -85,B 0,C 180,E1 -20913.675,E2 -20913.675} C_VEL
LIN {X 0,Y 283.288,Z 329.614,A -85,B 0,C 180,E1 -20915.353,E2 -20915.353} C_VEL
LIN {X 0,Y 274.469,Z 431.622,A -85,B 0,C 180,E1 -20917.894,E2 -20917.894} C_VEL
LIN {X 0,Y 271.861,Z 448.571,A -85,B 0,C 180,E1 -20918.507,E2 -20918.507} C_VEL
LIN {X 0,Y 268.435,Z 464.504,A -85,B 0,C 180,E1 -20919.288,E2 -20919.288} C_VEL
LIN {X 0,Y 264.039,Z 480.851,A -85,B 0,C 180,E1 -20920.368,E2 -20920.368} C_VEL
LIN {X 0,Y 259.538,Z 495.008,A -85,B 0,C 180,E1 -20921.579,E2 -20921.579} C_VEL
LIN {X 0,Y 254.086,Z 509.676,A -85,B 0,C 180,E1 -20923.154,E2 -20923.154} C_VEL
LIN {X 0,Y 248.823,Z 522.034,A -85,B 0,C 180,E1 -20924.795,E2 -20924.795} C_VEL
LIN {X 0,Y 242.433,Z 535.779,A -85,B 0,C 180,E1 -20927.06,E2 -20927.06} C_VEL
LIN {X 0,Y 235.935,Z 548.376,A -85,B 0,C 180,E1 -20929.619,E2 -20929.619} C_VEL
LIN {X 0,Y 230.06,Z 559.139,A -85,B 0,C 180,E1 -20932.342,E2 -20932.342} C_VEL
LIN {X 0,Y 224.044,Z 569.542,A -85,B 0,C 180,E1 -20935.624,E2 -20935.624} C_VEL
LIN {X 0,Y 218.791,Z 578.335,A -85,B 0,C 180,E1 -20939.074,E2 -20939.074} C_VEL
LIN {X 0,Y 214.35,Z 585.78,A -85,B 0,C 180,E1 -20942.677,E2 -20942.677} C_VEL
LIN {X 0,Y 210.781,Z 591.924,A -85,B 0,C 180,E1 -20946.416,E2 -20946.416} C_VEL
LIN {X 0,Y 208.043,Z 596.925,A -85,B 0,C 180,E1 -20950.257,E2 -20950.257} C_VEL
LIN {X 0,Y 206.089,Z 600.892,A -85,B 0,C 180,E1 -20954.169,E2 -20954.169} C_VEL
LIN {X 0,Y 204.855,Z 603.798,A -85,B 0,C 180,E1 -20958.122,E2 -20958.122} C_VEL
LIN {X 0,Y 204.351,Z 605.771,A -85,B 0,C 180,E1 -20962.094,E2 -20962.094} C_VEL
LIN {X 0,Y 204.295,Z 606.722,A -85,B 0,C 180,E1 -20966.055,E2 -20966.055} C_VEL
LIN {X 0,Y 204.479,Z 606.748,A -85,B 0,C 180,E1 -20970.001,E2 -20970.001} C_VEL
LIN {X 0,Y 204.345,Z 605.639,A -85,B 0,C 180,E1 -20974.145,E2 -20974.145} C_VEL
LIN {X 0,Y 204.365,Z 603.725,A -85,B 0,C 180,E1 -20977.907,E2 -20977.907} C_VEL
LIN {X 0,Y 204.846,Z 600.62,A -85,B 0,C 180,E1 -20981.88,E2 -20981.88} C_VEL
LIN {X 0,Y 206.025,Z 596.499,A -85,B 0,C 180,E1 -20985.837,E2 -20985.837} C_VEL
LIN {X 0,Y 207.799,Z 591.115,A -85,B 0,C 180,E1 -20989.768,E2 -20989.768} C_VEL
LIN {X 0,Y 210.379,Z 584.515,A -85,B 0,C 180,E1 -20993.633,E2 -20993.633} C_VEL
LIN {X 0,Y 213.712,Z 576.545,A -85,B 0,C 180,E1 -20997.413,E2 -20997.413} C_VEL
LIN {X 0,Y 217.956,Z 566.942,A -85,B 0,C 180,E1 -21001.059,E2 -21001.059} C_VEL
LIN {X 0,Y 222.343,Z 556.979,A -85,B 0,C 180,E1 -21004.129,E2 -21004.129} C_VEL
LIN {X 0,Y 226.439,Z 547.131,A -85,B 0,C 180,E1 -21006.688,E2 -21006.688} C_VEL
LIN {X 0,Y 231.486,Z 534.733,A -85,B 0,C 180,E1 -21009.329,E2 -21009.329} C_VEL
LIN {X 0,Y 236.558,Z 521.174,A -85,B 0,C 180,E1 -21011.663,E2 -21011.663} C_VEL
LIN {X 0,Y 241.094,Z 507.846,A -85,B 0,C 180,E1 -21013.525,E2 -21013.525} C_VEL
LIN {X 0,Y 245.397,Z 493.666,A -85,B 0,C 180,E1 -21015.139,E2 -21015.139} C_VEL
LIN {X 0,Y 249.346,Z 478.422,A -85,B 0,C 180,E1 -21016.534,E2 -21016.534} C_VEL
LIN {X 0,Y 252.924,Z 461.499,A -85,B 0,C 180,E1 -21017.717,E2 -21017.717} C_VEL
LIN {X 0,Y 255.779,Z 444.721,A -85,B 0,C 180,E1 -21018.541,E2 -21018.541} C_VEL
LIN {X 0,Y 257.612,Z 428.484,A -85,B 0,C 180,E1 -21019.11,E2 -21019.11} C_VEL
LIN {X 0,Y 264.936,Z 321.109,A -85,B 0,C 180,E1 -21021.921,E2 -21021.921} C_VEL
LIN {X 0,Y 257.284,Z 305.107,A -85,B 0,C 180,E1 -21024.457,E2 -21024.457} C_VEL
LIN {X 0,Y 250.235,Z 291.724,A -85,B 0,C 180,E1 -21026.973,E2 -21026.973} C_VEL
LIN {X 0,Y 245.213,Z 282.938,A -85,B 0,C 180,E1 -21028.884,E2 -21028.884} C_VEL
LIN {X 0,Y 241.807,Z 277.271,A -85,B 0,C 180,E1 -21030.254,E2 -21030.254} C_VEL
LIN {X 0,Y 234.574,Z 267.151,A -85,B 0,C 180,E1 -21033.294,E2 -21033.294} C_VEL
LIN {X 0,Y 230.858,Z 262.188,A -85,B 0,C 180,E1 -21035.014,E2 -21035.014} C_VEL
LIN {X 0,Y 227.708,Z 257.996,A -85,B 0,C 180,E1 -21036.559,E2 -21036.559} C_VEL
LIN {X 0,Y 224.277,Z 253.643,A -85,B 0,C 180,E1 -21038.335,E2 -21038.335} C_VEL
LIN {X 0,Y 221.464,Z 250.312,A -85,B 0,C 180,E1 -21039.887,E2 -21039.887} C_VEL
LIN {X 0,Y 220.314,Z 248.614,A -85,B 0,C 180,E1 -21040.582,E2 -21040.582} C_VEL
LIN {X 0,Y 217.553,Z 245.728,A -85,B 0,C 180,E1 -21042.243,E2 -21042.243} C_VEL
LIN {X 0,Y 216.091,Z 243.374,A -85,B 0,C 180,E1 -21043.223,E2 -21043.223} C_VEL
LIN {X 0,Y 213.324,Z 240.984,A -85,B 0,C 180,E1 -21045.024,E2 -21045.024} C_VEL
LIN {X 0,Y 211.855,Z 238.089,A -85,B 0,C 180,E1 -21046.206,E2 -21046.206} C_VEL
LIN {X 0,Y 208.856,Z 236.011,A -85,B 0,C 180,E1 -21048.475,E2 -21048.475} C_VEL
LIN {X 0,Y 207.511,Z 233.758,A -85,B 0,C 180,E1 -21049.696,E2 -21049.696} C_VEL
LIN {X 0,Y 207.081,Z 231.961,A -85,B 0,C 180,E1 -21050.23,E2 -21050.23} C_VEL
LIN {X 0,Y 207.054,Z 231.974,A -85,B 0,C 180,E1 -21054.156,E2 -21054.156} C_VEL
LIN {X 0,Y 207.378,Z 231.905,A -85,B 0,C 180,E1 -21058.058,E2 -21058.058} C_VEL
LIN {X 0,Y 207.511,Z 231.919,A -85,B 0,C 180,E1 -21060,E2 -21060} C_VEL
LIN {X 0,Y 207.38,Z 231.966,A -85,B 0,C 180,E1 -21061.942,E2 -21061.942} C_VEL
LIN {X 0,Y 207.141,Z 231.989,A -85,B 0,C 180,E1 -21067.8,E2 -21067.8} C_VEL
LIN {X 0,Y 206.924,Z 231.987,A -85,B 0,C 180,E1 -21071.758,E2 -21071.758} C_VEL
LIN {X 0,Y 206.868,Z 232.025,A -85,B 0,C 180,E1 -21075.771,E2 -21075.771} C_VEL
LIN {X 0,Y 206.784,Z 232.009,A -85,B 0,C 180,E1 -21079.869,E2 -21079.869} C_VEL
LIN {X 0,Y 206.764,Z 232.017,A -85,B 0,C 180,E1 -21084.072,E2 -21084.072} C_VEL
LIN {X 0,Y 206.745,Z 232.043,A -85,B 0,C 180,E1 -21088.419,E2 -21088.419} C_VEL
LIN {X 0,Y 206.702,Z 232.023,A -85,B 0,C 180,E1 -21092.957,E2 -21092.957} C_VEL
LIN {X 0,Y 206.716,Z 232.173,A -85,B 0,C 180,E1 -21096.057,E2 -21096.057} C_VEL
LIN {X 0,Y 207.59,Z 234.741,A -85,B 0,C 180,E1 -21097.012,E2 -21097.012} C_VEL
LIN {X 0,Y 209.703,Z 237.001,A -85,B 0,C 180,E1 -21098.752,E2 -21098.752} C_VEL
LIN {X 0,Y 211.657,Z 238.157,A -85,B 0,C 180,E1 -21100.186,E2 -21100.186} C_VEL
LIN {X 0,Y 213.164,Z 241.017,A -85,B 0,C 180,E1 -21101.4,E2 -21101.4} C_VEL
LIN {X 0,Y 215.815,Z 243.357,A -85,B 0,C 180,E1 -21103.146,E2 -21103.146} C_VEL
LIN {X 0,Y 216.447,Z 244.012,A -85,B 0,C 180,E1 -21103.548,E2 -21103.548} C_VEL
LIN {X 0,Y 218.564,Z 247.229,A -85,B 0,C 180,E1 -21104.943,E2 -21104.943} C_VEL
LIN {X 0,Y 220.832,Z 249.404,A -85,B 0,C 180,E1 -21106.26,E2 -21106.26} C_VEL
LIN {X 0,Y 223.394,Z 252.882,A -85,B 0,C 180,E1 -21107.727,E2 -21107.727} C_VEL
LIN {X 0,Y 225.115,Z 254.686,A -85,B 0,C 180,E1 -21108.622,E2 -21108.622} C_VEL
LIN {X 0,Y 228.174,Z 258.593,A -85,B 0,C 180,E1 -21110.201,E2 -21110.201} C_VEL
LIN {X 0,Y 233.269,Z 265.48,A -85,B 0,C 180,E1 -21112.635,E2 -21112.635} C_VEL
LIN {X 0,Y 238.947,Z 273.191,A -85,B 0,C 180,E1 -21115.104,E2 -21115.104} C_VEL
LIN {X 0,Y 246.123,Z 283.574,A -85,B 0,C 180,E1 -21117.944,E2 -21117.944} C_VEL
LIN {X 0,Y 255.324,Z 298.247,A -85,B 0,C 180,E1 -21121.237,E2 -21121.237} C_VEL
LIN {X 0,Y 263.321,Z 312.179,A -85,B 0,C 180,E1 -21123.844,E2 -21123.844} C_VEL
LIN {X 0,Y 265.027,Z 315.319,A -85,B 0,C 180,E1 -21124.371,E2 -21124.371} C_VEL
LIN {X 0,Y 257.776,Z 420.729,A -85,B 0,C 180,E1 -21127.138,E2 -21127.138} C_VEL
LIN {X 0,Y 255.749,Z 437.445,A -85,B 0,C 180,E1 -21127.799,E2 -21127.799} C_VEL
LIN {X 0,Y 253.02,Z 453.831,A -85,B 0,C 180,E1 -21128.726,E2 -21128.726} C_VEL
LIN {X 0,Y 249.9,Z 468.826,A -85,B 0,C 180,E1 -21129.848,E2 -21129.848} C_VEL
LIN {X 0,Y 246.141,Z 483.761,A -85,B 0,C 180,E1 -21131.263,E2 -21131.263} C_VEL
LIN {X 0,Y 241.987,Z 497.663,A -85,B 0,C 180,E1 -21132.902,E2 -21132.902} C_VEL
LIN {X 0,Y 237.273,Z 511.887,A -85,B 0,C 180,E1 -21134.979,E2 -21134.979} C_VEL
LIN {X 0,Y 232.331,Z 525.076,A -85,B 0,C 180,E1 -21137.331,E2 -21137.331} C_VEL
LIN {X 0,Y 227.829,Z 536.374,A -85,B 0,C 180,E1 -21139.783,E2 -21139.783} C_VEL
LIN {X 0,Y 222.988,Z 547.606,A -85,B 0,C 180,E1 -21142.757,E2 -21142.757} C_VEL
LIN {X 0,Y 218.723,Z 557.217,A -85,B 0,C 180,E1 -21145.859,E2 -21145.859} C_VEL
LIN {X 0,Y 214.55,Z 566.521,A -85,B 0,C 180,E1 -21149.53,E2 -21149.53} C_VEL
LIN {X 0,Y 211.186,Z 574.222,A -85,B 0,C 180,E1 -21153.286,E2 -21153.286} C_VEL
LIN {X 0,Y 208.125,Z 581.428,A -85,B 0,C 180,E1 -21157.762,E2 -21157.762} C_VEL
LIN {X 0,Y 206.27,Z 586.389,A -85,B 0,C 180,E1 -21161.795,E2 -21161.795} C_VEL
LIN {X 0,Y 204.89,Z 590.454,A -85,B 0,C 180,E1 -21166.171,E2 -21166.171} C_VEL
LIN {X 0,Y 204.173,Z 593.037,A -85,B 0,C 180,E1 -21170.133,E2 -21170.133} C_VEL
LIN {X 0,Y 203.854,Z 594.654,A -85,B 0,C 180,E1 -21174.437,E2 -21174.437} C_VEL
LIN {X 0,Y 203.927,Z 595.186,A -85,B 0,C 180,E1 -21178.847,E2 -21178.847} C_VEL
LIN {X 0,Y 204.473,Z 594.515,A -85,B 0,C 180,E1 -21183.362,E2 -21183.362} C_VEL
LIN {X 0,Y 205.745,Z 592.363,A -85,B 0,C 180,E1 -21188.219,E2 -21188.219} C_VEL
LIN {X 0,Y 207.676,Z 589.132,A -85,B 0,C 180,E1 -21192.595,E2 -21192.595} C_VEL
LIN {X 0,Y 210.621,Z 584.265,A -85,B 0,C 180,E1 -21197.229,E2 -21197.229} C_VEL
LIN {X 0,Y 214.725,Z 577.757,A -85,B 0,C 180,E1 -21201.767,E2 -21201.767} C_VEL
LIN {X 0,Y 218.838,Z 571.335,A -85,B 0,C 180,E1 -21205.243,E2 -21205.243} C_VEL
LIN {X 0,Y 223.946,Z 563.158,A -85,B 0,C 180,E1 -21208.777,E2 -21208.777} C_VEL
LIN {X 0,Y 229.228,Z 554.478,A -85,B 0,C 180,E1 -21211.816,E2 -21211.816} C_VEL
LIN {X 0,Y 234.924,Z 544.582,A -85,B 0,C 180,E1 -21214.649,E2 -21214.649} C_VEL
LIN {X 0,Y 240.409,Z 534.294,A -85,B 0,C 180,E1 -21217.048,E2 -21217.048} C_VEL
LIN {X 0,Y 246.705,Z 521.604,A -85,B 0,C 180,E1 -21219.473,E2 -21219.473} C_VEL
LIN {X 0,Y 252.141,Z 509.462,A -85,B 0,C 180,E1 -21221.382,E2 -21221.382} C_VEL
LIN {X 0,Y 257.822,Z 494.956,A -85,B 0,C 180,E1 -21223.227,E2 -21223.227} C_VEL
LIN {X 0,Y 262.774,Z 480.445,A -85,B 0,C 180,E1 -21224.685,E2 -21224.685} C_VEL
LIN {X 0,Y 267.187,Z 465.087,A -85,B 0,C 180,E1 -21225.913,E2 -21225.913} C_VEL
LIN {X 0,Y 270.735,Z 449.81,A -85,B 0,C 180,E1 -21226.878,E2 -21226.878} C_VEL
LIN {X 0,Y 273.673,Z 433.769,A -85,B 0,C 180,E1 -21227.615,E2 -21227.615} C_VEL
LIN {X 0,Y 275.773,Z 416.576,A -85,B 0,C 180,E1 -21228.161,E2 -21228.161} C_VEL
LIN {X 0,Y 283.48,Z 325.352,A -85,B 0,C 180,E1 -21230.445,E2 -21230.445} C_VEL
LIN {X 0,Y 278.466,Z 315.662,A -85,B 0,C 180,E1 -21233.083,E2 -21233.083} C_VEL
LIN {X 0,Y 275.245,Z 310.025,A -85,B 0,C 180,E1 -21234.988,E2 -21234.988} C_VEL
LIN {X 0,Y 271.629,Z 303.844,A -85,B 0,C 180,E1 -21237.444,E2 -21237.444} C_VEL
LIN {X 0,Y 269.527,Z 300.522,A -85,B 0,C 180,E1 -21239.092,E2 -21239.092} C_VEL
LIN {X 0,Y 267.062,Z 296.526,A -85,B 0,C 180,E1 -21241.363,E2 -21241.363} C_VEL
LIN {X 0,Y 264.571,Z 292.357,A -85,B 0,C 180,E1 -21244.316,E2 -21244.316} C_VEL
LIN {X 0,Y 262.448,Z 290.318,A -85,B 0,C 180,E1 -21247.784,E2 -21247.784} C_VEL
LIN {X 0,Y 261.672,Z 287.534,A -85,B 0,C 180,E1 -21251.275,E2 -21251.275} C_VEL
LIN {X 0,Y 261.568,Z 287.382,A -85,B 0,C 180,E1 -21252.367,E2 -21252.367} C_VEL
LIN {X 0,Y 261.514,Z 287.786,A -85,B 0,C 180,E1 -21253.22,E2 -21253.22} C_VEL
LIN {X 0,Y 261.446,Z 288.884,A -85,B 0,C 180,E1 -21254.047,E2 -21254.047} C_VEL
LIN {X 0,Y 261.302,Z 292.265,A -85,B 0,C 180,E1 -21255.626,E2 -21255.626} C_VEL
LIN {X 0,Y 261.462,Z 296.725,A -85,B 0,C 180,E1 -21257.604,E2 -21257.604} C_VEL
LIN {X 0,Y 261.924,Z 298.295,A -85,B 0,C 180,E1 -21258.863,E2 -21258.863} C_VEL
LIN {X 0,Y 263.169,Z 299.598,A -85,B 0,C 180,E1 -21260.826,E2 -21260.826} C_VEL
LIN {X 0,Y 265.358,Z 303.188,A -85,B 0,C 180,E1 -21263.595,E2 -21263.595} C_VEL
LIN {X 0,Y 268.653,Z 308.655,A -85,B 0,C 180,E1 -21266.72,E2 -21266.72} C_VEL
LIN {X 0,Y 270.938,Z 313.189,A -85,B 0,C 180,E1 -21268.568,E2 -21268.568} C_VEL
LIN {X 0,Y 273.829,Z 318.962,A -85,B 0,C 180,E1 -21270.581,E2 -21270.581} C_VEL
LIN {X 0,Y 277.81,Z 328.241,A -85,B 0,C 180,E1 -21273.074,E2 -21273.074} C_VEL
LIN {X 0,Y 279.668,Z 332.868,A -85,B 0,C 180,E1 -21274.145,E2 -21274.145} C_VEL
LIN {X 0,Y 270.845,Z 431.641,A -85,B 0,C 180,E1 -21276.609,E2 -21276.609} C_VEL
LIN {X 0,Y 268.065,Z 449.106,A -85,B 0,C 180,E1 -21277.241,E2 -21277.241} C_VEL
LIN {X 0,Y 264.387,Z 465.432,A -85,B 0,C 180,E1 -21278.049,E2 -21278.049} C_VEL
LIN {X 0,Y 260.168,Z 480.494,A -85,B 0,C 180,E1 -21279.048,E2 -21279.048} C_VEL
LIN {X 0,Y 255.53,Z 494.626,A -85,B 0,C 180,E1 -21280.252,E2 -21280.252} C_VEL
LIN {X 0,Y 249.878,Z 509.29,A -85,B 0,C 180,E1 -21281.814,E2 -21281.814} C_VEL
LIN {X 0,Y 244.457,Z 521.676,A -85,B 0,C 180,E1 -21283.456,E2 -21283.456} C_VEL
LIN {X 0,Y 238.293,Z 534.489,A -85,B 0,C 180,E1 -21285.537,E2 -21285.537} C_VEL
LIN {X 0,Y 232.459,Z 545.513,A -85,B 0,C 180,E1 -21287.726,E2 -21287.726} C_VEL
LIN {X 0,Y 226.136,Z 556.561,A -85,B 0,C 180,E1 -21290.424,E2 -21290.424} C_VEL
LIN {X 0,Y 219.729,Z 567.357,A -85,B 0,C 180,E1 -21293.722,E2 -21293.722} C_VEL
LIN {X 0,Y 213.953,Z 576.502,A -85,B 0,C 180,E1 -21297.181,E2 -21297.181} C_VEL
LIN {X 0,Y 208.818,Z 584.593,A -85,B 0,C 180,E1 -21301.051,E2 -21301.051} C_VEL
LIN {X 0,Y 204.199,Z 591.967,A -85,B 0,C 180,E1 -21305.607,E2 -21305.607} C_VEL
LIN {X 0,Y 201.284,Z 596.904,A -85,B 0,C 180,E1 -21309.565,E2 -21309.565} C_VEL
LIN {X 0,Y 199.18,Z 600.84,A -85,B 0,C 180,E1 -21313.605,E2 -21313.605} C_VEL
LIN {X 0,Y 197.834,Z 603.682,A -85,B 0,C 180,E1 -21317.694,E2 -21317.694} C_VEL
LIN {X 0,Y 197.278,Z 605.626,A -85,B 0,C 180,E1 -21321.808,E2 -21321.808} C_VEL
LIN {X 0,Y 197.204,Z 606.561,A -85,B 0,C 180,E1 -21326.257,E2 -21326.257} C_VEL
LIN {X 0,Y 197.379,Z 606.529,A -85,B 0,C 180,E1 -21330.001,E2 -21330.001} C_VEL
LIN {X 0,Y 197.248,Z 605.448,A -85,B 0,C 180,E1 -21334.087,E2 -21334.087} C_VEL
LIN {X 0,Y 197.289,Z 603.426,A -85,B 0,C 180,E1 -21338.193,E2 -21338.193} C_VEL
LIN {X 0,Y 197.825,Z 600.264,A -85,B 0,C 180,E1 -21342.308,E2 -21342.308} C_VEL
LIN {X 0,Y 199.118,Z 596.087,A -85,B 0,C 180,E1 -21346.402,E2 -21346.402} C_VEL
LIN {X 0,Y 201.027,Z 590.667,A -85,B 0,C 180,E1 -21350.463,E2 -21350.463} C_VEL
LIN {X 0,Y 203.778,Z 584,A -85,B 0,C 180,E1 -21354.448,E2 -21354.448} C_VEL
LIN {X 0,Y 207.313,Z 575.956,A -85,B 0,C 180,E1 -21358.334,E2 -21358.334} C_VEL
LIN {X 0,Y 211.786,Z 566.308,A -85,B 0,C 180,E1 -21362.07,E2 -21362.07} C_VEL
LIN {X 0,Y 215.713,Z 557.781,A -85,B 0,C 180,E1 -21364.761,E2 -21364.761} C_VEL
LIN {X 0,Y 219.919,Z 548.107,A -85,B 0,C 180,E1 -21367.386,E2 -21367.386} C_VEL
LIN {X 0,Y 225.505,Z 534.844,A -85,B 0,C 180,E1 -21370.292,E2 -21370.292} C_VEL
LIN {X 0,Y 230.637,Z 521.63,A -85,B 0,C 180,E1 -21372.615,E2 -21372.615} C_VEL
LIN {X 0,Y 235.431,Z 508.066,A -85,B 0,C 180,E1 -21374.548,E2 -21374.548} C_VEL
LIN {X 0,Y 239.865,Z 493.978,A -85,B 0,C 180,E1 -21376.179,E2 -21376.179} C_VEL
LIN {X 0,Y 243.924,Z 478.805,A -85,B 0,C 180,E1 -21377.588,E2 -21377.588} C_VEL
LIN {X 0,Y 247.322,Z 463.311,A -85,B 0,C 180,E1 -21378.699,E2 -21378.699} C_VEL
LIN {X 0,Y 250.233,Z 447.18,A -85,B 0,C 180,E1 -21379.544,E2 -21379.544} C_VEL
LIN {X 0,Y 252.413,Z 429.903,A -85,B 0,C 180,E1 -21380.179,E2 -21380.179} C_VEL
LIN {X 0,Y 259.963,Z 323.817,A -85,B 0,C 180,E1 -21382.971,E2 -21382.971} C_VEL
LIN {X 0,Y 252.982,Z 309.031,A -85,B 0,C 180,E1 -21385.406,E2 -21385.406} C_VEL
LIN {X 0,Y 246.061,Z 295.707,A -85,B 0,C 180,E1 -21387.982,E2 -21387.982} C_VEL
LIN {X 0,Y 239.302,Z 283.829,A -85,B 0,C 180,E1 -21390.716,E2 -21390.716} C_VEL
LIN {X 0,Y 231.934,Z 273.227,A -85,B 0,C 180,E1 -21393.921,E2 -21393.921} C_VEL
LIN {X 0,Y 225.019,Z 263.884,A -85,B 0,C 180,E1 -21397.316,E2 -21397.316} C_VEL
LIN {X 0,Y 221.89,Z 259.858,A -85,B 0,C 180,E1 -21398.996,E2 -21398.996} C_VEL
LIN {X 0,Y 219.001,Z 256.265,A -85,B 0,C 180,E1 -21400.667,E2 -21400.667} C_VEL
LIN {X 0,Y 217.964,Z 254.871,A -85,B 0,C 180,E1 -21401.303,E2 -21401.303} C_VEL
LIN {X 0,Y 215.203,Z 251.732,A -85,B 0,C 180,E1 -21403.03,E2 -21403.03} C_VEL
LIN {X 0,Y 213.923,Z 249.81,A -85,B 0,C 180,E1 -21403.907,E2 -21403.907} C_VEL
LIN {X 0,Y 211.263,Z 247.23,A -85,B 0,C 180,E1 -21405.737,E2 -21405.737} C_VEL
LIN {X 0,Y 209.82,Z 244.553,A -85,B 0,C 180,E1 -21406.933,E2 -21406.933} C_VEL
LIN {X 0,Y 207.127,Z 242.58,A -85,B 0,C 180,E1 -21409.043,E2 -21409.043} C_VEL
LIN {X 0,Y 205.498,Z 239.802,A -85,B 0,C 180,E1 -21410.583,E2 -21410.583} C_VEL
LIN {X 0,Y 205.09,Z 238.792,A -85,B 0,C 180,E1 -21411.025,E2 -21411.025} C_VEL
LIN {X 0,Y 202.118,Z 237.049,A -85,B 0,C 180,E1 -21413.887,E2 -21413.887} C_VEL
LIN {X 0,Y 200.623,Z 234.963,A -85,B 0,C 180,E1 -21415.731,E2 -21415.731} C_VEL
LIN {X 0,Y 200.11,Z 232.805,A -85,B 0,C 180,E1 -21416.728,E2 -21416.728} C_VEL
LIN {X 0,Y 200.476,Z 232.793,A -85,B 0,C 180,E1 -21420,E2 -21420} C_VEL
LIN {X 0,Y 200.024,Z 232.851,A -85,B 0,C 180,E1 -21424.03,E2 -21424.03} C_VEL
LIN {X 0,Y 200.089,Z 232.871,A -85,B 0,C 180,E1 -21428.077,E2 -21428.077} C_VEL
LIN {X 0,Y 199.875,Z 232.864,A -85,B 0,C 180,E1 -21432.179,E2 -21432.179} C_VEL
LIN {X 0,Y 199.806,Z 232.895,A -85,B 0,C 180,E1 -21436.343,E2 -21436.343} C_VEL
LIN {X 0,Y 199.701,Z 232.899,A -85,B 0,C 180,E1 -21440.605,E2 -21440.605} C_VEL
LIN {X 0,Y 199.673,Z 232.893,A -85,B 0,C 180,E1 -21444.984,E2 -21444.984} C_VEL
LIN {X 0,Y 199.669,Z 232.929,A -85,B 0,C 180,E1 -21449.439,E2 -21449.439} C_VEL
LIN {X 0,Y 200.262,Z 234.978,A -85,B 0,C 180,E1 -21450.442,E2 -21450.442} C_VEL
LIN {X 0,Y 202.064,Z 237.387,A -85,B 0,C 180,E1 -21452.621,E2 -21452.621} C_VEL
LIN {X 0,Y 204.946,Z 239.09,A -85,B 0,C 180,E1 -21455.416,E2 -21455.416} C_VEL
LIN {X 0,Y 205.976,Z 241.453,A -85,B 0,C 180,E1 -21456.511,E2 -21456.511} C_VEL
LIN {X 0,Y 208.311,Z 243.891,A -85,B 0,C 180,E1 -21458.479,E2 -21458.479} C_VEL
LIN {X 0,Y 209.732,Z 244.797,A -85,B 0,C 180,E1 -21459.544,E2 -21459.544} C_VEL
LIN {X 0,Y 211.758,Z 248.12,A -85,B 0,C 180,E1 -21461.172,E2 -21461.172} C_VEL
LIN {X 0,Y 214.445,Z 250.631,A -85,B 0,C 180,E1 -21462.982,E2 -21462.982} C_VEL
LIN {X 0,Y 216.966,Z 254.147,A -85,B 0,C 180,E1 -21464.644,E2 -21464.644} C_VEL
LIN {X 0,Y 218.635,Z 255.819,A -85,B 0,C 180,E1 -21465.644,E2 -21465.644} C_VEL
LIN {X 0,Y 221.498,Z 259.564,A -85,B 0,C 180,E1 -21467.32,E2 -21467.32} C_VEL
LIN {X 0,Y 223.017,Z 261.356,A -85,B 0,C 180,E1 -21468.145,E2 -21468.145} C_VEL
LIN {X 0,Y 227.172,Z 266.881,A -85,B 0,C 180,E1 -21470.321,E2 -21470.321} C_VEL
LIN {X 0,Y 232.955,Z 274.631,A -85,B 0,C 180,E1 -21473.059,E2 -21473.059} C_VEL
LIN {X 0,Y 240.878,Z 286.07,A -85,B 0,C 180,E1 -21476.435,E2 -21476.435} C_VEL
LIN {X 0,Y 249.557,Z 299.853,A -85,B 0,C 180,E1 -21479.745,E2 -21479.745} C_VEL
LIN {X 0,Y 255.734,Z 310.446,A -85,B 0,C 180,E1 -21481.899,E2 -21481.899} C_VEL
LIN {X 0,Y 259.989,Z 318.21,A -85,B 0,C 180,E1 -21483.306,E2 -21483.306} C_VEL
LIN {X 0,Y 253.691,Z 408.212,A -85,B 0,C 180,E1 -21485.664,E2 -21485.664} C_VEL
LIN {X 0,Y 251.978,Z 427.342,A -85,B 0,C 180,E1 -21486.254,E2 -21486.254} C_VEL
LIN {X 0,Y 249.516,Z 444.541,A -85,B 0,C 180,E1 -21487.05,E2 -21487.05} C_VEL
LIN {X 0,Y 246.594,Z 459.981,A -85,B 0,C 180,E1 -21488.033,E2 -21488.033} C_VEL
LIN {X 0,Y 243.132,Z 474.782,A -85,B 0,C 180,E1 -21489.261,E2 -21489.261} C_VEL
LIN {X 0,Y 238.899,Z 490.186,A -85,B 0,C 180,E1 -21490.896,E2 -21490.896} C_VEL
LIN {X 0,Y 234.234,Z 504.49,A -85,B 0,C 180,E1 -21492.765,E2 -21492.765} C_VEL
LIN {X 0,Y 229.007,Z 518.85,A -85,B 0,C 180,E1 -21495.106,E2 -21495.106} C_VEL
LIN {X 0,Y 224.008,Z 531.341,A -85,B 0,C 180,E1 -21497.616,E2 -21497.616} C_VEL
LIN {X 0,Y 219.243,Z 542.359,A -85,B 0,C 180,E1 -21500.311,E2 -21500.311} C_VEL
LIN {X 0,Y 214.491,Z 552.742,A -85,B 0,C 180,E1 -21503.414,E2 -21503.414} C_VEL
LIN {X 0,Y 209.754,Z 562.817,A -85,B 0,C 180,E1 -21507.119,E2 -21507.119} C_VEL
LIN {X 0,Y 205.836,Z 571.243,A -85,B 0,C 180,E1 -21510.978,E2 -21510.978} C_VEL
LIN {X 0,Y 202.708,Z 578.257,A -85,B 0,C 180,E1 -21514.972,E2 -21514.972} C_VEL
LIN {X 0,Y 199.851,Z 585.093,A -85,B 0,C 180,E1 -21520.051,E2 -21520.051} C_VEL
LIN {X 0,Y 198.226,Z 589.373,A -85,B 0,C 180,E1 -21524.369,E2 -21524.369} C_VEL
LIN {X 0,Y 197.251,Z 592.467,A -85,B 0,C 180,E1 -21528.702,E2 -21528.702} C_VEL
LIN {X 0,Y 196.809,Z 594.508,A -85,B 0,C 180,E1 -21533.128,E2 -21533.128} C_VEL
LIN {X 0,Y 196.758,Z 595.349,A -85,B 0,C 180,E1 -21537.667,E2 -21537.667} C_VEL
LIN {X 0,Y 197.198,Z 595.042,A -85,B 0,C 180,E1 -21542.315,E2 -21542.315} C_VEL
LIN {X 0,Y 198.253,Z 593.51,A -85,B 0,C 180,E1 -21547.058,E2 -21547.058} C_VEL
LIN {X 0,Y 200.186,Z 590.602,A -85,B 0,C 180,E1 -21551.838,E2 -21551.838} C_VEL
LIN {X 0,Y 202.998,Z 586.192,A -85,B 0,C 180,E1 -21556.637,E2 -21556.637} C_VEL
LIN {X 0,Y 205.966,Z 581.714,A -85,B 0,C 180,E1 -21560.294,E2 -21560.294} C_VEL
LIN {X 0,Y 210.699,Z 574.788,A -85,B 0,C 180,E1 -21564.676,E2 -21564.676} C_VEL
LIN {X 0,Y 216.255,Z 566.556,A -85,B 0,C 180,E1 -21568.669,E2 -21568.669} C_VEL
LIN {X 0,Y 222.343,Z 557.095,A -85,B 0,C 180,E1 -21572.255,E2 -21572.255} C_VEL
LIN {X 0,Y 228.322,Z 547.281,A -85,B 0,C 180,E1 -21575.233,E2 -21575.233} C_VEL
LIN {X 0,Y 234.877,Z 535.782,A -85,B 0,C 180,E1 -21578.058,E2 -21578.058} C_VEL
LIN {X 0,Y 241.368,Z 523.375,A -85,B 0,C 180,E1 -21580.502,E2 -21580.502} C_VEL
LIN {X 0,Y 247.6,Z 510.012,A -85,B 0,C 180,E1 -21582.632,E2 -21582.632} C_VEL
LIN {X 0,Y 253.705,Z 494.964,A -85,B 0,C 180,E1 -21584.549,E2 -21584.549} C_VEL
LIN {X 0,Y 258.891,Z 480.287,A -85,B 0,C 180,E1 -21586.013,E2 -21586.013} C_VEL
LIN {X 0,Y 263.11,Z 466.155,A -85,B 0,C 180,E1 -21587.146,E2 -21587.146} C_VEL
LIN {X 0,Y 266.66,Z 451.703,A -85,B 0,C 180,E1 -21588.079,E2 -21588.079} C_VEL
LIN {X 0,Y 269.737,Z 435.481,A -85,B 0,C 180,E1 -21588.847,E2 -21588.847} C_VEL
LIN {X 0,Y 272.018,Z 418.441,A -85,B 0,C 180,E1 -21589.394,E2 -21589.394} C_VEL
LIN {X 0,Y 279.906,Z 329.09,A -85,B 0,C 180,E1 -21591.619,E2 -21591.619} C_VEL
LIN {X 0,Y 275.318,Z 319.987,A -85,B 0,C 180,E1 -21594.231,E2 -21594.231} C_VEL
LIN {X 0,Y 271.194,Z 312.669,A -85,B 0,C 180,E1 -21596.958,E2 -21596.958} C_VEL
LIN {X 0,Y 268.294,Z 307.51,A -85,B 0,C 180,E1 -21599.264,E2 -21599.264} C_VEL
LIN {X 0,Y 265.794,Z 303.573,A -85,B 0,C 180,E1 -21601.61,E2 -21601.61} C_VEL
LIN {X 0,Y 264.725,Z 301.846,A -85,B 0,C 180,E1 -21602.782,E2 -21602.782} C_VEL
LIN {X 0,Y 263.388,Z 299.294,A -85,B 0,C 180,E1 -21604.591,E2 -21604.591} C_VEL
LIN {X 0,Y 261.343,Z 297.123,A -85,B 0,C 180,E1 -21608.162,E2 -21608.162} C_VEL
LIN {X 0,Y 260.717,Z 294.57,A -85,B 0,C 180,E1 -21611.317,E2 -21611.317} C_VEL
LIN {X 0,Y 260.608,Z 294.516,A -85,B 0,C 180,E1 -21613.227,E2 -21613.227} C_VEL
LIN {X 0,Y 260.669,Z 295.124,A -85,B 0,C 180,E1 -21614.48,E2 -21614.48} C_VEL
LIN {X 0,Y 261.924,Z 298.295,A -85,B 0,C 180,E1 -21618.863,E2 -21618.863} C_VEL
LIN {X 0,Y 262.294,Z 299.562,A -85,B 0,C 180,E1 -21619.676,E2 -21619.676} C_VEL
LIN {X 0,Y 262.656,Z 303.524,A -85,B 0,C 180,E1 -21620.854,E2 -21620.854} C_VEL
LIN {X 0,Y 263.081,Z 307.776,A -85,B 0,C 180,E1 -21622.013,E2 -21622.013} C_VEL
LIN {X 0,Y 263.625,Z 309.473,A -85,B 0,C 180,E1 -21622.8,E2 -21622.8} C_VEL
LIN {X 0,Y 264.661,Z 311.1,A -85,B 0,C 180,E1 -21623.944,E2 -21623.944} C_VEL
LIN {X 0,Y 267.06,Z 315.267,A -85,B 0,C 180,E1 -21626.264,E2 -21626.264} C_VEL
LIN {X 0,Y 270.07,Z 321.432,A -85,B 0,C 180,E1 -21628.745,E2 -21628.745} C_VEL
LIN {X 0,Y 272.81,Z 327.69,A -85,B 0,C 180,E1 -21630.707,E2 -21630.707} C_VEL
LIN {X 0,Y 276.177,Z 336.129,A -85,B 0,C 180,E1 -21632.871,E2 -21632.871} C_VEL
LIN {X 0,Y 276.133,Z 337.962,A -85,B 0,C 180,E1 -21632.97,E2 -21632.97} C_VEL
LIN {X 0,Y 267.417,Z 431.312,A -85,B 0,C 180,E1 -21635.28,E2 -21635.28} C_VEL
LIN {X 0,Y 264.545,Z 448.844,A -85,B 0,C 180,E1 -21635.907,E2 -21635.907} C_VEL
LIN {X 0,Y 260.772,Z 465.157,A -85,B 0,C 180,E1 -21636.701,E2 -21636.701} C_VEL
LIN {X 0,Y 256.44,Z 480.231,A -85,B 0,C 180,E1 -21637.69,E2 -21637.69} C_VEL
LIN {X 0,Y 251.64,Z 494.38,A -85,B 0,C 180,E1 -21638.877,E2 -21638.877} C_VEL
LIN {X 0,Y 245.823,Z 509.017,A -85,B 0,C 180,E1 -21640.432,E2 -21640.432} C_VEL
LIN {X 0,Y 240.227,Z 521.365,A -85,B 0,C 180,E1 -21642.069,E2 -21642.069} C_VEL
LIN {X 0,Y 233.294,Z 535.123,A -85,B 0,C 180,E1 -21644.32,E2 -21644.32} C_VEL
